  MoveL 9043 to (510.41, 540.16, 160) mm, rotated rx 180 ry 0 rz 160 deg; joints [10.972, 56.166, -5.021, -142.378, 57.459, 157.483]
  Set speed (17.1 mm/s)
  Call Extruder(1063.40800)
  MoveL 9044 to (509.43, 540.4, 160) mm, rotated rx -180 ry 0 rz 160 deg; joints [11.024, 56.007, -4.715, -142.378, 57.595, 157.558]
  Set speed (17.1 mm/s)
  Call Extruder(1069.01822)
  MoveL 9045 to (507.77, 540.76, 160) mm, rotated rx 180 ry 0 rz 160 deg; joints [11.105, 55.733, -4.19, -142.385, 57.825, 157.692]
  Call Extruder(1074.68107)
  MoveL 9046 to (506.08, 541.04, 160) mm, rotated rx 180 ry 0 rz 160 deg; joints [11.18, 55.455, -3.655, -142.401, 58.057, 157.833]
  Call Extruder(1080.09055)
  MoveL 9047 to (504.45, 541.25, 160) mm, rotated rx 180 ry 0 rz 160 deg; joints [11.245, 55.187, -3.141, -142.425, 58.276, 157.973]
  Set speed (17.1 mm/s)
  Call Extruder(1085.82019)
  MoveL 9048 to (502.71, 541.4, 160) mm, rotated rx -180 ry 0 rz 160 deg; joints [11.305, 54.901, -2.592, -142.458, 58.507, 158.127]
  Set speed (17.1 mm/s)
  Call Extruder(1091.48567)
  MoveL 9049 to (501, 541.48, 160) mm, rotated rx -180 ry 0 rz 160 deg; joints [11.357, 54.617, -2.047, -142.499, 58.734, 158.284]
  Set speed (17.1 mm/s)
  Call Extruder(1096.89132)
  MoveL 9050 to (499.36, 541.49, 160) mm, rotated rx -180 ry 0 rz 160 deg; joints [11.398, 54.346, -1.526, -142.546, 58.947, 158.438]
  Set speed (10.0 mm/s)
  MoveL 9051 to (499.36, 541.49, 164) mm, rotated rx 180 ry 0 rz 160 deg; joints [11.398, 53.788, -1.416, -142.38, 58.592, 158.119]
  Set speed (120.0 mm/s)
  MoveL 9052 to (500.97, 540.23, 164) mm, rotated rx -180 ry 0 rz 160 deg; joints [11.204, 54.015, -1.85, -142.513, 58.356, 158.081]
  Set speed (17.3 mm/s)
  Call Extruder(1102.39668)
  MoveL 9053 to (499.29, 540.24, 164) mm, rotated rx 180 ry 0 rz 160 deg; joints [11.246, 53.735, -1.315, -142.564, 58.573, 158.239]
  Call Extruder(1107.72599)
  MoveL 9054 to (497.66, 540.17, 164) mm, rotated rx 180 ry 0 rz 160 deg; joints [11.278, 53.463, -0.796, -142.62, 58.781, 158.397]
  Set speed (17.2 mm/s)
  Call Extruder(1113.18708)
  MoveL 9055 to (496, 540.04, 164) mm, rotated rx -180 ry 0 rz 160 deg; joints [11.303, 53.185, -0.265, -142.685, 58.991, 158.562]
  Call Extruder(1118.52641)
  MoveL 9056 to (494.38, 539.85, 164) mm, rotated rx -180 ry 0 rz 160 deg; joints [11.319, 52.913, 0.253, -142.758, 59.193, 158.727]
  Set speed (17.3 mm/s)
  Call Extruder(1123.71666)
  MoveL 9057 to (492.81, 539.59, 164) mm, rotated rx -180 ry 0 rz 160 deg; joints [11.326, 52.65, 0.755, -142.835, 59.387, 158.891]
  Call Extruder(1129.28278)
  MoveL 9058 to (491.14, 539.26, 164) mm, rotated rx -180 ry 0 rz 160 deg; joints [11.326, 52.369, 1.291, -142.926, 59.59, 159.07]
  Set speed (17.2 mm/s)
  Call Extruder(1134.66464)
  MoveL 9059 to (489.55, 538.86, 164) mm, rotated rx 180 ry 0 rz 160 deg; joints [11.317, 52.1, 1.806, -143.022, 59.782, 159.246]
  Set speed (17.2 mm/s)
  Call Extruder(1139.87147)
  MoveL 9060 to (488.02, 538.42, 164) mm, rotated rx -180 ry 0 rz 160 deg; joints [11.299, 51.841, 2.299, -143.123, 59.964, 159.419]
  Set speed (17.2 mm/s)
  Call Extruder(1145.48231)
  MoveL 9061 to (486.39, 537.87, 164) mm, rotated rx 180 ry 0 rz 160 deg; joints [11.271, 51.565, 2.826, -143.24, 60.155, 159.607]
  Set speed (17.2 mm/s)
  Call Extruder(1150.53984)
  MoveL 9062 to (484.95, 537.32, 164) mm, rotated rx 180 ry 0 rz 160 deg; joints [11.238, 51.319, 3.296, -143.352, 60.322, 159.779]
  Set speed (17.2 mm/s)
  Call Extruder(1155.86729)
  MoveL 9063 to (483.45, 536.68, 164) mm, rotated rx 180 ry 0 rz 160 deg; joints [11.195, 51.063, 3.784, -143.478, 60.494, 159.962]
  Set speed (17.3 mm/s)
  Call Extruder(1159.63536)
  MoveL 9064 to (482.41, 536.2, 164) mm, rotated rx 180 ry 0 rz 160 deg; joints [11.159, 50.884, 4.127, -143.571, 60.613, 160.092]
  Call Extruder(1164.11046)
  MoveL 9065 to (481.19, 535.58, 164) mm, rotated rx 180 ry 0 rz 160 deg; joints [11.11, 50.674, 4.527, -143.688, 60.75, 160.247]
  Set speed (17.3 mm/s)
  Call Extruder(1166.72011)
  MoveL 9066 to (480.49, 535.2, 164) mm, rotated rx 180 ry 0 rz 160 deg; joints [11.079, 50.553, 4.758, -143.757, 60.828, 160.338]
  Call Extruder(1169.33186)
  MoveL 9067 to (479.79, 534.8, 164) mm, rotated rx 180 ry 0 rz 160 deg; joints [11.046, 50.433, 4.987, -143.829, 60.905, 160.429]
  Set speed (17.2 mm/s)
  Call Extruder(1172.31752)
  MoveL 9068 to (479.01, 534.33, 164) mm, rotated rx 180 ry 0 rz 160 deg; joints [11.005, 50.297, 5.246, -143.913, 60.991, 160.534]
  Set speed (17.3 mm/s)
  Call Extruder(1175.98709)
  MoveL 9069 to (478.06, 533.74, 164) mm, rotated rx 180 ry 0 rz 160 deg; joints [10.952, 50.132, 5.561, -144.019, 61.095, 160.662]
  Call Extruder(1180.42460)
  MoveL 9070 to (476.94, 532.98, 164) mm, rotated rx 180 ry 0 rz 160 deg; joints [10.882, 49.936, 5.935, -144.153, 61.216, 160.818]
  Set speed (17.2 mm/s)
  Call Extruder(1183.09673)
  MoveL 9071 to (476.27, 532.5, 164) mm, rotated rx -180 ry 0 rz 160 deg; joints [10.836, 49.82, 6.157, -144.235, 61.287, 160.912]
  Set speed (17.2 mm/s)
  Call Extruder(1185.65152)
  MoveL 9072 to (475.65, 532.04, 164) mm, rotated rx -180 ry 0 rz 160 deg; joints [10.791, 49.71, 6.367, -144.316, 61.353, 161.002]
  Set speed (17.2 mm/s)
  Call Extruder(1188.25211)
  MoveL 9073 to (475.02, 531.55, 164) mm, rotated rx -180 ry 0 rz 160 deg; joints [10.744, 49.6, 6.578, -144.399, 61.419, 161.093]
  Set speed (17.2 mm/s)
  Call Extruder(1191.21831)
  MoveL 9074 to (474.31, 530.98, 164) mm, rotated rx 180 ry 0 rz 160 deg; joints [10.687, 49.475, 6.815, -144.496, 61.493, 161.197]
  Set speed (17.2 mm/s)
  Call Extruder(1193.83711)
  MoveL 9075 to (473.7, 530.46, 164) mm, rotated rx 180 ry 0 rz 160 deg; joints [10.634, 49.367, 7.021, -144.584, 61.556, 161.289]
  Set speed (17.2 mm/s)
  Call Extruder(1196.39663)
  MoveL 9076 to (473.11, 529.95, 164) mm, rotated rx 180 ry 0 rz 160 deg; joints [10.581, 49.263, 7.22, -144.671, 61.616, 161.379]
  Set speed (17.2 mm/s)
  Call Extruder(1199.09717)
  MoveL 9077 to (472.51, 529.39, 164) mm, rotated rx -180 ry 0 rz 160 deg; joints [10.522, 49.155, 7.427, -144.764, 61.678, 161.473]
  Call Extruder(1201.94180)
  MoveL 9078 to (471.88, 528.79, 164) mm, rotated rx -180 ry 0 rz 160 deg; joints [10.459, 49.042, 7.641, -144.865, 61.741, 161.572]
  Set speed (17.2 mm/s)
  Call Extruder(1207.42131)
  MoveL 9079 to (470.71, 527.59, 164) mm, rotated rx 180 ry 0 rz 160 deg; joints [10.329, 48.832, 8.043, -145.063, 61.857, 161.763]
  Set speed (17.2 mm/s)
  Call Extruder(1209.85171)
  MoveL 9080 to (470.2, 527.05, 164) mm, rotated rx 180 ry 0 rz 160 deg; joints [10.27, 48.74, 8.218, -145.153, 61.906, 161.847]
  Set speed (17.2 mm/s)
  Call Extruder(1212.71687)
  MoveL 9081 to (469.62, 526.39, 164) mm, rotated rx 180 ry 0 rz 160 deg; joints [10.197, 48.635, 8.419, -145.26, 61.963, 161.946]
  Call Extruder(1215.30637)
  MoveL 9082 to (469.11, 525.79, 164) mm, rotated rx 180 ry 0 rz 160 deg; joints [10.129, 48.541, 8.597, -145.359, 62.011, 162.035]
  Set speed (17.2 mm/s)
  Call Extruder(1217.99933)
  MoveL 9083 to (468.59, 525.15, 164) mm, rotated rx -180 ry 0 rz 160 deg; joints [10.057, 48.446, 8.78, -145.463, 62.061, 162.127]
  Set speed (17.2 mm/s)
  Call Extruder(1220.64109)
  MoveL 9084 to (468.09, 524.52, 164) mm, rotated rx -180 ry 0 rz 160 deg; joints [9.984, 48.354, 8.955, -145.566, 62.107, 162.217]
  Set speed (17.2 mm/s)
  Call Extruder(1223.38075)
  MoveL 9085 to (467.58, 523.85, 164) mm, rotated rx -180 ry 0 rz 160 deg; joints [9.907, 48.261, 9.132, -145.675, 62.153, 162.31]
  Set speed (17.2 mm/s)
  Call Extruder(1226.20172)
  MoveL 9086 to (467.08, 523.15, 164) mm, rotated rx -180 ry 0 rz 160 deg; joints [9.825, 48.168, 9.311, -145.788, 62.199, 162.406]
  Set speed (17.3 mm/s)
  Call Extruder(1228.73103)
  MoveL 9087 to (466.64, 522.51, 164) mm, rotated rx 180 ry 0 rz 160 deg; joints [9.75, 48.086, 9.467, -145.891, 62.238, 162.491]
  Set speed (17.3 mm/s)
  Call Extruder(1231.44468)
  MoveL 9088 to (466.19, 521.82, 164) mm, rotated rx 180 ry 0 rz 160 deg; joints [9.668, 48, 9.631, -146.003, 62.278, 162.581]
  Set speed (17.2 mm/s)
  Call Extruder(1234.06972)
  MoveL 9089 to (465.76, 521.14, 164) mm, rotated rx 180 ry 0 rz 160 deg; joints [9.587, 47.919, 9.786, -146.112, 62.315, 162.668]
  Call Extruder(1236.82307)
  MoveL 9090 to (465.32, 520.42, 164) mm, rotated rx -180 ry 0 rz 160 deg; joints [9.499, 47.836, 9.944, -146.228, 62.351, 162.759]
  Set speed (17.3 mm/s)
  Call Extruder(1239.50905)
  MoveL 9091 to (464.92, 519.71, 164) mm, rotated rx -180 ry 0 rz 160 deg; joints [9.413, 47.757, 10.094, -146.342, 62.385, 162.847]
  Set speed (17.2 mm/s)
  Call Extruder(1242.30123)
  MoveL 9092 to (464.5, 518.96, 164) mm, rotated rx -180 ry 0 rz 160 deg; joints [9.321, 47.678, 10.246, -146.461, 62.418, 162.938]
  Set speed (17.2 mm/s)
  Call Extruder(1244.88259)
  MoveL 9093 to (464.14, 518.26, 164) mm, rotated rx 180 ry 0 rz 160 deg; joints [9.235, 47.607, 10.381, -146.573, 62.447, 163.021]
  Set speed (17.3 mm/s)
  Call Extruder(1247.52606)
  MoveL 9094 to (463.78, 517.54, 164) mm, rotated rx 180 ry 0 rz 160 deg; joints [9.145, 47.536, 10.516, -146.689, 62.474, 163.106]
  Set speed (17.2 mm/s)
  Call Extruder(1252.88420)
  MoveL 9095 to (463.09, 516.05, 164) mm, rotated rx -180 ry 0 rz 160 deg; joints [8.958, 47.4, 10.777, -146.925, 62.524, 163.276]
  Set speed (17.2 mm/s)
  Call Extruder(1258.25337)
  MoveL 9096 to (462.47, 514.53, 164) mm, rotated rx -180 ry 0 rz 160 deg; joints [8.765, 47.273, 11.019, -147.166, 62.566, 163.442]
  Set speed (17.2 mm/s)
  Call Extruder(1263.67576)
  MoveL 9097 to (461.91, 512.98, 164) mm, rotated rx 180 ry 0 rz 160 deg; joints [8.565, 47.154, 11.245, -147.413, 62.599, 163.608]
  Call Extruder(1269.06660)
  MoveL 9098 to (461.41, 511.41, 164) mm, rotated rx 180 ry 0 rz 160 deg; joints [8.361, 47.046, 11.452, -147.66, 62.625, 163.768]
  Set speed (17.2 mm/s)
  Call Extruder(1274.56925)
  MoveL 9099 to (460.97, 509.78, 164) mm, rotated rx 180 ry 0 rz 160 deg; joints [8.148, 46.946, 11.642, -147.916, 62.643, 163.929]
  Set speed (17.2 mm/s)
  Call Extruder(1279.89206)
  MoveL 9100 to (460.6, 508.2, 164) mm, rotated rx -180 ry 0 rz 160 deg; joints [7.938, 46.86, 11.807, -148.165, 62.651, 164.08]
  Set speed (17.3 mm/s)
  Call Extruder(1285.41223)
  MoveL 9101 to (460.29, 506.54, 164) mm, rotated rx -180 ry 0 rz 160 deg; joints [7.717, 46.781, 11.958, -148.424, 62.652, 164.233]
  Call Extruder(1290.88446)
  MoveL 9102 to (460.06, 504.88, 164) mm, rotated rx -180 ry 0 rz 160 deg; joints [7.493, 46.714, 12.086, -148.683, 62.644, 164.38]
  Set speed (17.2 mm/s)
  Call Extruder(1296.18613)
  MoveL 9103 to (459.89, 503.27, 164) mm, rotated rx -180 ry 0 rz 160 deg; joints [7.274, 46.659, 12.191, -148.934, 62.627, 164.518]
  Set speed (17.3 mm/s)
  Call Extruder(1301.69852)
  MoveL 9104 to (459.79, 501.59, 164) mm, rotated rx 180 ry 0 rz 160 deg; joints [7.044, 46.613, 12.279, -149.195, 62.602, 164.657]
  Set speed (17.2 mm/s)
  Call Extruder(1306.85050)
  MoveL 9105 to (459.75, 500.02, 164) mm, rotated rx -180 ry 0 rz 160 deg; joints [6.827, 46.579, 12.342, -149.438, 62.571, 164.783]
  Call Extruder(1311.56706)
  MoveL 9106 to (459.78, 498.58, 164) mm, rotated rx 180 ry 0 rz 160 deg; joints [6.628, 46.559, 12.381, -149.66, 62.535, 164.894]
  Call Extruder(1316.68940)
  MoveL 9107 to (459.87, 497.01, 164) mm, rotated rx 180 ry 0 rz 160 deg; joints [6.41, 46.545, 12.408, -149.9, 62.489, 165.01]
  Set speed (17.3 mm/s)
  Call Extruder(1321.58133)
  MoveL 9108 to (460.01, 495.52, 164) mm, rotated rx -180 ry 0 rz 160 deg; joints [6.202, 46.541, 12.415, -150.128, 62.439, 165.117]
  Set speed (17.3 mm/s)
  Call Extruder(1326.10523)
  MoveL 9109 to (460.19, 494.15, 164) mm, rotated rx 180 ry 0 rz 160 deg; joints [6.01, 46.546, 12.406, -150.337, 62.386, 165.212]
  Set speed (17.3 mm/s)
  Call Extruder(1331.17816)
  MoveL 9110 to (460.44, 492.62, 164) mm, rotated rx -180 ry 0 rz 160 deg; joints [5.794, 46.56, 12.379, -150.569, 62.32, 165.314]
  Set speed (17.3 mm/s)
  Call Extruder(1335.86329)
  MoveL 9111 to (460.73, 491.22, 164) mm, rotated rx -180 ry 0 rz 160 deg; joints [5.596, 46.582, 12.337, -150.78, 62.252, 165.403]
  Set speed (17.2 mm/s)
  Call Extruder(1340.95386)
  MoveL 9112 to (461.1, 489.71, 164) mm, rotated rx 180 ry 0 rz 160 deg; joints [5.382, 46.615, 12.275, -151.007, 62.173, 165.496]
  Set speed (17.2 mm/s)
  Call Extruder(1345.56843)
  MoveL 9113 to (461.48, 488.35, 164) mm, rotated rx 180 ry 0 rz 160 deg; joints [5.19, 46.653, 12.202, -151.209, 62.094, 165.576]
  Set speed (17.2 mm/s)
  Call Extruder(1350.72526)
  MoveL 9114 to (461.97, 486.85, 164) mm, rotated rx 180 ry 0 rz 160 deg; joints [4.976, 46.705, 12.103, -151.431, 62, 165.66]
  Set speed (17.2 mm/s)
  Call Extruder(1355.73817)
  MoveL 9115 to (462.5, 485.41, 164) mm, rotated rx 180 ry 0 rz 160 deg; joints [4.771, 46.765, 11.989, -151.642, 61.901, 165.737]
  Call Extruder(1360.34080)
  MoveL 9116 to (463.03, 484.11, 164) mm, rotated rx 180 ry 0 rz 160 deg; joints [4.585, 46.828, 11.869, -151.832, 61.805, 165.802]
  Set speed (17.3 mm/s)
  Call Extruder(1365.27188)
  MoveL 9117 to (463.65, 482.74, 164) mm, rotated rx 180 ry 0 rz 160 deg; joints [4.389, 46.904, 11.723, -152.03, 61.696, 165.867]
  Set speed (17.2 mm/s)
  Call Extruder(1369.73169)
  MoveL 9118 to (464.26, 481.52, 164) mm, rotated rx 180 ry 0 rz 160 deg; joints [4.214, 46.98, 11.578, -152.205, 61.592, 165.922]
  Set speed (17.2 mm/s)
  Call Extruder(1374.93959)
  MoveL 9119 to (465.01, 480.12, 164) mm, rotated rx 180 ry 0 rz 160 deg; joints [4.014, 47.078, 11.391, -152.404, 61.465, 165.98]
  Set speed (17.2 mm/s)
  Call Extruder(1379.75206)
  MoveL 9120 to (465.76, 478.85, 164) mm, rotated rx 180 ry 0 rz 160 deg; joints [3.833, 47.176, 11.203, -152.581, 61.342, 166.029]
  Call Extruder(1384.92062)
  MoveL 9121 to (466.62, 477.52, 164) mm, rotated rx 180 ry 0 rz 160 deg; joints [3.643, 47.291, 10.984, -152.766, 61.204, 166.076]
  Call Extruder(1389.45717)
  MoveL 9122 to (467.41, 476.39, 164) mm, rotated rx -180 ry 0 rz 160 deg; joints [3.481, 47.399, 10.778, -152.921, 61.077, 166.111]
  Set speed (17.2 mm/s)
  Call Extruder(1394.19668)
  MoveL 9123 to (468.28, 475.23, 164) mm, rotated rx 180 ry 0 rz 160 deg; joints [3.315, 47.519, 10.549, -153.077, 60.94, 166.144]
  Call Extruder(1399.13732)
  MoveL 9124 to (469.23, 474.06, 164) mm, rotated rx 180 ry 0 rz 160 deg; joints [3.148, 47.652, 10.295, -153.233, 60.792, 166.172]
  Set speed (17.3 mm/s)
  Call Extruder(1403.98459)
  MoveL 9125 to (470.21, 472.94, 164) mm, rotated rx -180 ry 0 rz 160 deg; joints [2.988, 47.79, 10.032, -153.379, 60.642, 166.194]
  Set speed (17.3 mm/s)
  Call Extruder(1408.72195)
  MoveL 9126 to (471.2, 471.89, 164) mm, rotated rx 180 ry 0 rz 160 deg; joints [2.838, 47.932, 9.762, -153.514, 60.491, 166.21]
  Set speed (17.3 mm/s)
  Call Extruder(1413.62945)
  MoveL 9127 to (472.27, 470.84, 164) mm, rotated rx 180 ry 0 rz 160 deg; joints [2.688, 48.086, 9.468, -153.646, 60.33, 166.222]
  Set speed (17.2 mm/s)
  Call Extruder(1418.25129)
  MoveL 9128 to (473.31, 469.88, 164) mm, rotated rx 180 ry 0 rz 160 deg; joints [2.552, 48.237, 9.179, -153.763, 60.175, 166.227]
  Call Extruder(1423.26639)
  MoveL 9129 to (474.48, 468.88, 164) mm, rotated rx 180 ry 0 rz 160 deg; joints [2.411, 48.408, 8.853, -153.882, 60.002, 166.227]
  Call Extruder(1428.06443)
  MoveL 9130 to (475.63, 467.97, 164) mm, rotated rx 180 ry 0 rz 160 deg; joints [2.282, 48.577, 8.529, -153.988, 59.832, 166.221]
  Call Extruder(1433.02690)
  MoveL 9131 to (476.86, 467.08, 164) mm, rotated rx 180 ry 0 rz 160 deg; joints [2.155, 48.76, 8.181, -154.088, 59.653, 166.209]
  Set speed (17.3 mm/s)
  Call Extruder(1437.79644)
  MoveL 9132 to (478.06, 466.26, 164) mm, rotated rx 180 ry 0 rz 160 deg; joints [2.04, 48.941, 7.835, -154.176, 59.478, 166.191]
  Set speed (17.3 mm/s)
  Call Extruder(1442.40095)
  MoveL 9133 to (479.26, 465.52, 164) mm, rotated rx -180 ry 0 rz 160 deg; joints [1.934, 49.121, 7.492, -154.252, 59.305, 166.169]
  Set speed (17.3 mm/s)
  Call Extruder(1447.50015)
  MoveL 9134 to (480.61, 464.74, 164) mm, rotated rx -180 ry 0 rz 160 deg; joints [1.825, 49.326, 7.1, -154.329, 59.111, 166.139]
  Set speed (17.2 mm/s)
  Call Extruder(1453.20412)
  MoveL 9135 to (482.15, 463.93, 164) mm, rotated rx 180 ry 0 rz 160 deg; joints [1.711, 49.562, 6.65, -154.401, 58.891, 166.097]
  Set speed (17.2 mm/s)
  Call Extruder(1457.17333)
  MoveL 9136 to (483.25, 463.41, 164) mm, rotated rx 180 ry 0 rz 160 deg; joints [1.638, 49.73, 6.329, -154.444, 58.735, 166.062]
  Set speed (17.2 mm/s)
  Call Extruder(1461.95242)
  MoveL 9137 to (484.59, 462.83, 164) mm, rotated rx -180 ry 0 rz 160 deg; joints [1.556, 49.937, 5.934, -154.488, 58.545, 166.016]
  Set speed (17.3 mm/s)
  Call Extruder(1466.98216)
  MoveL 9138 to (486.02, 462.27, 164) mm, rotated rx -180 ry 0 rz 160 deg; joints [1.477, 50.16, 5.509, -154.525, 58.344, 165.961]
  Set speed (17.2 mm/s)
  Call Extruder(1471.84329)
  MoveL 9139 to (487.42, 461.77, 164) mm, rotated rx -180 ry 0 rz 160 deg; joints [1.408, 50.379, 5.09, -154.55, 58.147, 165.902]
  Call Extruder(1476.74031)
  MoveL 9140 to (488.85, 461.33, 164) mm, rotated rx 180 ry 0 rz 160 deg; joints [1.346, 50.604, 4.661, -154.567, 57.947, 165.836]
  Set speed (17.3 mm/s)
  Call Extruder(1481.51368)
  MoveL 9141 to (490.26, 460.96, 164) mm, rotated rx -180 ry 0 rz 160 deg; joints [1.292, 50.827, 4.235, -154.573, 57.751, 165.766]
  Set speed (17.3 mm/s)
  Call Extruder(1486.28147)
  MoveL 9142 to (491.68, 460.63, 164) mm, rotated rx 180 ry 0 rz 160 deg; joints [1.245, 51.053, 3.804, -154.571, 57.554, 165.69]
  Set speed (17.3 mm/s)
  Call Extruder(1490.95394)
  MoveL 9143 to (493.08, 460.36, 164) mm, rotated rx 180 ry 0 rz 160 deg; joints [1.206, 51.277, 3.375, -154.56, 57.36, 165.61]
  Set speed (17.3 mm/s)
  Call Extruder(1496.06278)
  MoveL 9144 to (494.63, 460.12, 164) mm, rotated rx 180 ry 0 rz 160 deg; joints [1.171, 51.526, 2.902, -154.538, 57.148, 165.517]
  Set speed (17.2 mm/s)
  Call Extruder(1500.87565)
  MoveL 9145 to (496.09, 459.95, 164) mm, rotated rx 180 ry 0 rz 160 deg; joints [1.146, 51.762, 2.451, -154.507, 56.948, 165.423]
  Set speed (17.2 mm/s)
  Call Extruder(1505.77291)
  MoveL 9146 to (497.58, 459.83, 164) mm, rotated rx -180 ry 0 rz 160 deg; joints [1.127, 52.005, 1.987, -154.468, 56.744, 165.321]
  Set speed (17.3 mm/s)
  Call Extruder(1510.56917)
  MoveL 9147 to (499.05, 459.77, 164) mm, rotated rx -180 ry 0 rz 160 deg; joints [1.115, 52.244, 1.53, -154.419, 56.544, 165.216]
  Set speed (17.3 mm/s)
  Call Extruder(1515.26906)
  MoveL 9148 to (500.48, 459.76, 164) mm, rotated rx 180 ry 0 rz 160 deg; joints [1.11, 52.48, 1.079, -154.363, 56.35, 165.108]
  Call Extruder(1520.34091)
  MoveL 9149 to (502.03, 459.81, 164) mm, rotated rx -180 ry 0 rz 160 deg; joints [1.113, 52.737, 0.59, -154.293, 56.14, 164.985]
  Set speed (17.3 mm/s)
  Call Extruder(1525.13170)
  MoveL 9150 to (503.49, 459.91, 164) mm, rotated rx 180 ry 0 rz 160 deg; joints [1.122, 52.98, 0.125, -154.217, 55.944, 164.863]
  Set speed (17.2 mm/s)
  Call Extruder(1529.97241)
  MoveL 9151 to (504.96, 460.07, 164) mm, rotated rx -180 ry 0 rz 160 deg; joints [1.138, 53.226, -0.344, -154.133, 55.746, 164.735]
  Set speed (17.2 mm/s)
  Call Extruder(1534.57519)
  MoveL 9152 to (506.36, 460.26, 164) mm, rotated rx -180 ry 0 rz 160 deg; joints [1.159, 53.461, -0.792, -154.044, 55.561, 164.608]
  Set speed (17.2 mm/s)
  Call Extruder(1539.34961)
  MoveL 9153 to (507.79, 460.52, 164) mm, rotated rx 180 ry 0 rz 160 deg; joints [1.188, 53.704, -1.256, -153.944, 55.37, 164.472]
  Set speed (17.3 mm/s)
  Call Extruder(1544.52807)
  MoveL 9154 to (509.34, 460.86, 164) mm, rotated rx -180 ry 0 rz 160 deg; joints [1.226, 53.968, -1.759, -153.827, 55.165, 164.318]
  Set speed (17.3 mm/s)
  Call Extruder(1549.38509)
  MoveL 9155 to (510.78, 461.23, 164) mm, rotated rx 180 ry 0 rz 160 deg; joints [1.268, 54.214, -2.23, -153.708, 54.975, 164.169]
  Set speed (17.3 mm/s)
  Call Extruder(1554.03460)
  MoveL 9156 to (512.14, 461.63, 164) mm, rotated rx 180 ry 0 rz 160 deg; joints [1.315, 54.45, -2.679, -153.586, 54.796, 164.021]
  Set speed (17.3 mm/s)
  Call Extruder(1558.96594)
  MoveL 9157 to (513.57, 462.12, 164) mm, rotated rx 180 ry 0 rz 160 deg; joints [1.37, 54.698, -3.153, -153.449, 54.61, 163.86]
  Call Extruder(1563.55660)
  MoveL 9158 to (514.88, 462.61, 164) mm, rotated rx -180 ry 0 rz 160 deg; joints [1.428, 54.928, -3.591, -153.315, 54.439, 163.706]
  Set speed (17.3 mm/s)
  Call Extruder(1568.65646)
  MoveL 9159 to (516.32, 463.22, 164) mm, rotated rx -180 ry 0 rz 160 deg; joints [1.498, 55.181, -4.075, -153.158, 54.254, 163.531]
  Call Extruder(0.00000)
  Set speed (17.3 mm/s)
  Call Extruder(4.61765)
  MoveL 9160 to (517.6, 463.81, 164) mm, rotated rx 180 ry 0 rz 160 deg; joints [1.567, 55.408, -4.509, -153.01, 54.089, 163.368]
  Set speed (17.3 mm/s)
  Call Extruder(9.77849)
  MoveL 9161 to (519.01, 464.53, 164) mm, rotated rx -180 ry 0 rz 160 deg; joints [1.65, 55.66, -4.988, -152.836, 53.91, 163.182]
  Set speed (17.3 mm/s)
  Call Extruder(14.71469)
  MoveL 9162 to (520.32, 465.27, 164) mm, rotated rx -180 ry 0 rz 160 deg; joints [1.735, 55.897, -5.44, -152.662, 53.744, 163]
  Call Extruder(19.28491)
  MoveL 9163 to (521.52, 466, 164) mm, rotated rx 180 ry 0 rz 160 deg; joints [1.819, 56.113, -5.853, -152.496, 53.594, 162.828]
  Set speed (17.3 mm/s)
  Call Extruder(24.21319)
  MoveL 9164 to (522.77, 466.82, 164) mm, rotated rx -180 ry 0 rz 160 deg; joints [1.915, 56.343, -6.292, -152.311, 53.437, 162.64]
  Set speed (17.3 mm/s)
  Call Extruder(28.89791)
  MoveL 9165 to (523.94, 467.66, 164) mm, rotated rx 180 ry 0 rz 160 deg; joints [2.011, 56.558, -6.702, -152.129, 53.293, 162.459]
  Set speed (17.3 mm/s)
  Call Extruder(33.82593)
  MoveL 9166 to (525.14, 468.57, 164) mm, rotated rx -180 ry 0 rz 160 deg; joints [2.116, 56.781, -7.126, -151.933, 53.147, 162.266]
  Set speed (17.2 mm/s)
  Call Extruder(38.75984)
  MoveL 9167 to (526.29, 469.54, 164) mm, rotated rx 180 ry 0 rz 160 deg; joints [2.227, 56.998, -7.541, -151.731, 53.007, 162.07]
  Set speed (17.3 mm/s)
  Call Extruder(43.43285)
  MoveL 9168 to (527.36, 470.49, 164) mm, rotated rx 180 ry 0 rz 160 deg; joints [2.336, 57.2, -7.926, -151.535, 52.88, 161.882]
  Set speed (17.3 mm/s)
  Call Extruder(48.58755)
  MoveL 9169 to (528.5, 471.58, 164) mm, rotated rx -180 ry 0 rz 160 deg; joints [2.462, 57.416, -8.339, -151.314, 52.746, 161.674]
  Call Extruder(53.66629)
  MoveL 9170 to (529.57, 472.71, 164) mm, rotated rx 180 ry 0 rz 160 deg; joints [2.59, 57.624, -8.735, -151.092, 52.622, 161.467]
  Set speed (17.3 mm/s)
  Call Extruder(56.40603)
  MoveL 9171 to (530.13, 473.33, 164) mm, rotated rx 180 ry 0 rz 160 deg; joints [2.661, 57.733, -8.944, -150.97, 52.558, 161.355]
  Set speed (17.2 mm/s)
  Call Extruder(59.26622)
  MoveL 9172 to (530.71, 473.99, 164) mm, rotated rx 180 ry 0 rz 160 deg; joints [2.737, 57.846, -9.158, -150.842, 52.493, 161.238]
  Set speed (17.2 mm/s)
  Call Extruder(61.81879)
  MoveL 9173 to (531.2, 474.59, 164) mm, rotated rx 180 ry 0 rz 160 deg; joints [2.805, 57.944, -9.345, -150.727, 52.437, 161.133]
  Set speed (17.2 mm/s)
  Call Extruder(64.41399)
  MoveL 9174 to (531.7, 475.21, 164) mm, rotated rx 180 ry 0 rz 160 deg; joints [2.876, 58.042, -9.532, -150.609, 52.383, 161.026]
  Call Extruder(67.13695)
  MoveL 9175 to (532.21, 475.87, 164) mm, rotated rx -180 ry 0 rz 160 deg; joints [2.951, 58.143, -9.725, -150.484, 52.327, 160.915]
  Set speed (17.2 mm/s)
  Call Extruder(69.90550)
  MoveL 9176 to (532.7, 476.55, 164) mm, rotated rx 180 ry 0 rz 160 deg; joints [3.029, 58.243, -9.917, -150.356, 52.274, 160.801]
  Call Extruder(72.52977)
  MoveL 9177 to (533.16, 477.21, 164) mm, rotated rx 180 ry 0 rz 160 deg; joints [3.104, 58.337, -10.095, -150.235, 52.225, 160.693]
  Call Extruder(78.09547)
  MoveL 9178 to (534.1, 478.63, 164) mm, rotated rx -180 ry 0 rz 160 deg; joints [3.266, 58.528, -10.459, -149.974, 52.128, 160.465]
  Set speed (17.2 mm/s)
  Call Extruder(82.89360)
  MoveL 9179 to (534.86, 479.88, 164) mm, rotated rx 180 ry 0 rz 160 deg; joints [3.409, 58.685, -10.759, -149.748, 52.053, 160.27]
  Set speed (17.2 mm/s)
  Call Extruder(87.82933)
  MoveL 9180 to (535.58, 481.2, 164) mm, rotated rx -180 ry 0 rz 160 deg; joints [3.559, 58.839, -11.052, -149.514, 51.983, 160.07]
  Set speed (17.2 mm/s)
  Call Extruder(91.41981)
  MoveL 9181 to (536.08, 482.18, 164) mm, rotated rx -180 ry 0 rz 160 deg; joints [3.67, 58.946, -11.256, -149.342, 51.938, 159.926]
  Set speed (17.2 mm/s)
  Call Extruder(94.08306)
  MoveL 9182 to (536.43, 482.91, 164) mm, rotated rx 180 ry 0 rz 160 deg; joints [3.754, 59.023, -11.402, -149.215, 51.907, 159.819]
  Set speed (17.2 mm/s)
  Call Extruder(96.97442)
  MoveL 9183 to (536.8, 483.71, 164) mm, rotated rx 180 ry 0 rz 160 deg; joints [3.845, 59.103, -11.556, -149.076, 51.876, 159.704]
  Set speed (17.2 mm/s)
  Call Extruder(102.36922)
  MoveL 9184 to (537.43, 485.23, 164) mm, rotated rx 180 ry 0 rz 160 deg; joints [4.018, 59.245, -11.827, -148.818, 51.826, 159.492]
  Set speed (17.2 mm/s)
  Call Extruder(107.64359)
  MoveL 9185 to (538, 486.74, 164) mm, rotated rx 180 ry 0 rz 160 deg; joints [4.19, 59.374, -12.073, -148.565, 51.786, 159.288]
  Set speed (17.2 mm/s)
  Call Extruder(113.16762)
  MoveL 9186 to (538.52, 488.35, 164) mm, rotated rx -180 ry 0 rz 160 deg; joints [4.373, 59.499, -12.31, -148.301, 51.755, 159.078]
  Set speed (17.3 mm/s)
  Call Extruder(118.32270)
  MoveL 9187 to (538.95, 489.87, 164) mm, rotated rx 180 ry 0 rz 160 deg; joints [4.547, 59.605, -12.512, -148.055, 51.736, 158.886]
  Call Extruder(123.83762)
  MoveL 9188 to (539.34, 491.51, 164) mm, rotated rx -180 ry 0 rz 160 deg; joints [4.734, 59.706, -12.706, -147.794, 51.726, 158.686]
  Set speed (17.3 mm/s)
  Call Extruder(129.16621)
  MoveL 9189 to (539.65, 493.11, 164) mm, rotated rx 180 ry 0 rz 160 deg; joints [4.917, 59.793, -12.871, -147.544, 51.726, 158.498]
  Set speed (17.2 mm/s)
  Call Extruder(134.76605)
  MoveL 9190 to (539.9, 494.8, 164) mm, rotated rx 180 ry 0 rz 160 deg; joints [5.111, 59.872, -13.023, -147.283, 51.737, 158.306]
  Set speed (17.2 mm/s)
  Call Extruder(140.24021)
  MoveL 9191 to (540.09, 496.46, 164) mm, rotated rx 180 ry 0 rz 160 deg; joints [5.302, 59.938, -13.147, -147.032, 51.758, 158.125]
  Set speed (17.3 mm/s)
  Call Extruder(145.52557)
  MoveL 9192 to (540.2, 498.07, 164) mm, rotated rx 180 ry 0 rz 160 deg; joints [5.488, 59.989, -13.245, -146.792, 51.789, 157.957]
  Set speed (17.3 mm/s)
  Call Extruder(150.71373)
  MoveL 9193 to (540.24, 499.66, 164) mm, rotated rx 180 ry 0 rz 160 deg; joints [5.672, 60.028, -13.32, -146.561, 51.828, 157.799]
  Set speed (17.3 mm/s)
  Call Extruder(156.30675)
  MoveL 9194 to (540.22, 501.37, 164) mm, rotated rx -180 ry 0 rz 160 deg; joints [5.87, 60.058, -13.376, -146.316, 51.881, 157.636]
  Set speed (17.2 mm/s)
  Call Extruder(161.64443)
  MoveL 9195 to (540.13, 503, 164) mm, rotated rx 180 ry 0 rz 160 deg; joints [6.06, 60.074, -13.407, -146.087, 51.941, 157.488]
  Call Extruder(167.06757)
  MoveL 9196 to (539.97, 504.65, 164) mm, rotated rx 180 ry 0 rz 160 deg; joints [6.253, 60.078, -13.414, -145.859, 52.012, 157.346]
  Set speed (17.3 mm/s)
  Call Extruder(172.42728)
  MoveL 9197 to (539.75, 506.27, 164) mm, rotated rx 180 ry 0 rz 160 deg; joints [6.443, 60.07, -13.399, -145.639, 52.092, 157.214]
  Call Extruder(177.54201)
  MoveL 9198 to (539.48, 507.81, 164) mm, rotated rx 180 ry 0 rz 160 deg; joints [6.625, 60.051, -13.362, -145.434, 52.177, 157.096]
  Set speed (17.3 mm/s)
  Call Extruder(183.16286)
  MoveL 9199 to (539.11, 509.49, 164) mm, rotated rx 180 ry 0 rz 160 deg; joints [6.824, 60.017, -13.298, -145.216, 52.28, 156.976]
  Set speed (17.3 mm/s)
  Call Extruder(189.03860)
  MoveL 9200 to (538.65, 511.23, 164) mm, rotated rx -180 ry 0 rz 160 deg; joints [7.032, 59.969, -13.207, -144.994, 52.396, 156.86]
  Set speed (17.3 mm/s)
  Call Extruder(193.69971)
  MoveL 9201 to (538.22, 512.59, 164) mm, rotated rx 180 ry 0 rz 160 deg; joints [7.195, 59.919, -13.111, -144.825, 52.498, 156.778]
  Set speed (17.3 mm/s)
  Call Extruder(199.08064)
  MoveL 9202 to (537.68, 514.14, 164) mm, rotated rx -180 ry 0 rz 160 deg; joints [7.383, 59.851, -12.982, -144.635, 52.623, 156.691]
  Set speed (17.2 mm/s)
  Call Extruder(204.66454)
  MoveL 9203 to (537.04, 515.72, 164) mm, rotated rx -180 ry 0 rz 160 deg; joints [7.576, 59.768, -12.825, -144.445, 52.76, 156.61]
  Set speed (17.3 mm/s)
  Call Extruder(209.82660)
  MoveL 9204 to (536.4, 517.16, 164) mm, rotated rx -180 ry 0 rz 160 deg; joints [7.753, 59.681, -12.658, -144.276, 52.894, 156.545]
  Set speed (17.3 mm/s)
  Call Extruder(212.76425)
  MoveL 9205 to (536.01, 517.97, 164) mm, rotated rx -180 ry 0 rz 160 deg; joints [7.853, 59.626, -12.554, -144.184, 52.974, 156.512]
  Set speed (17.2 mm/s)
  Call Extruder(215.42753)
  MoveL 9206 to (535.63, 518.7, 164) mm, rotated rx -180 ry 0 rz 160 deg; joints [7.942, 59.574, -12.453, -144.102, 53.049, 156.485]
  Set speed (17.2 mm/s)
  Call Extruder(218.19363)
  MoveL 9207 to (535.23, 519.44, 164) mm, rotated rx 180 ry 0 rz 160 deg; joints [8.035, 59.517, -12.345, -144.018, 53.128, 156.459]
  Call Extruder(220.87107)
  MoveL 9208 to (534.83, 520.15, 164) mm, rotated rx -180 ry 0 rz 160 deg; joints [8.124, 59.459, -12.235, -143.939, 53.206, 156.436]
  Call Extruder(223.51382)
  MoveL 9209 to (534.42, 520.85, 164) mm, rotated rx -180 ry 0 rz 160 deg; joints [8.212, 59.4, -12.121, -143.862, 53.284, 156.416]
  Set speed (17.2 mm/s)
  Call Extruder(226.01827)
  MoveL 9210 to (534.02, 521.5, 164) mm, rotated rx 180 ry 0 rz 160 deg; joints [8.294, 59.34, -12.008, -143.792, 53.361, 156.399]
  Call Extruder(230.46743)
  MoveL 9211 to (533.27, 522.63, 164) mm, rotated rx 180 ry 0 rz 160 deg; joints [8.439, 59.229, -11.797, -143.671, 53.5, 156.375]
  Set speed (17.3 mm/s)
  Call Extruder(234.10450)
  MoveL 9212 to (532.63, 523.55, 164) mm, rotated rx 180 ry 0 rz 160 deg; joints [8.556, 59.134, -11.615, -143.576, 53.616, 156.36]
  Set speed (17.3 mm/s)
  Call Extruder(236.82504)
  MoveL 9213 to (532.14, 524.22, 164) mm, rotated rx 180 ry 0 rz 160 deg; joints [8.642, 59.06, -11.473, -143.507, 53.705, 156.351]
  Set speed (17.2 mm/s)
  Call Extruder(239.67627)
  MoveL 9214 to (531.61, 524.91, 164) mm, rotated rx -180 ry 0 rz 160 deg; joints [8.732, 58.979, -11.319, -143.437, 53.8, 156.345]
  Call Extruder(242.36553)
  MoveL 9215 to (531.09, 525.55, 164) mm, rotated rx -180 ry 0 rz 160 deg; joints [8.816, 58.9, -11.168, -143.373, 53.891, 156.342]
  Set speed (17.2 mm/s)
  Call Extruder(246.49092)
  MoveL 9216 to (530.28, 526.51, 164) mm, rotated rx -180 ry 0 rz 160 deg; joints [8.943, 58.774, -10.929, -143.278, 54.034, 156.341]
  Set speed (17.2 mm/s)
  Call Extruder(251.80850)
  MoveL 9217 to (529.19, 527.71, 164) mm, rotated rx 180 ry 0 rz 160 deg; joints [9.103, 58.605, -10.606, -143.164, 54.221, 156.349]
  Set speed (17.2 mm/s)
  Call Extruder(255.86966)
  MoveL 9218 to (528.32, 528.59, 164) mm, rotated rx -180 ry 0 rz 160 deg; joints [9.223, 58.469, -10.347, -143.082, 54.368, 156.361]
  Set speed (17.3 mm/s)
  Call Extruder(258.43514)
  MoveL 9219 to (527.76, 529.14, 164) mm, rotated rx -180 ry 0 rz 160 deg; joints [9.297, 58.381, -10.178, -143.032, 54.462, 156.371]
  Set speed (17.3 mm/s)
  Call Extruder(261.06836)
  MoveL 9220 to (527.17, 529.69, 164) mm, rotated rx -180 ry 0 rz 160 deg; joints [9.373, 58.288, -10.002, -142.983, 54.559, 156.384]
  Call Extruder(263.80830)
  MoveL 9221 to (526.54, 530.25, 164) mm, rotated rx -180 ry 0 rz 160 deg; joints [9.451, 58.189, -9.814, -142.934, 54.661, 156.399]
  Set speed (17.2 mm/s)
  Call Extruder(266.42764)
  MoveL 9222 to (525.94, 530.77, 164) mm, rotated rx -180 ry 0 rz 160 deg; joints [9.524, 58.093, -9.63, -142.89, 54.76, 156.417]
  Call Extruder(269.15438)
  MoveL 9223 to (525.29, 531.3, 164) mm, rotated rx -180 ry 0 rz 160 deg; joints [9.599, 57.991, -9.435, -142.845, 54.864, 156.437]
  Set speed (17.2 mm/s)
  Call Extruder(272.04094)
  MoveL 9224 to (524.6, 531.85, 164) mm, rotated rx 180 ry 0 rz 160 deg; joints [9.677, 57.881, -9.225, -142.8, 54.975, 156.46]
  Set speed (17.2 mm/s)
  Call Extruder(274.48416)
  MoveL 9225 to (524.01, 532.3, 164) mm, rotated rx -180 ry 0 rz 160 deg; joints [9.742, 57.786, -9.043, -142.764, 55.07, 156.482]
  Set speed (17.3 mm/s)
  Call Extruder(277.27156)
  MoveL 9226 to (523.32, 532.8, 164) mm, rotated rx -180 ry 0 rz 160 deg; joints [9.815, 57.675, -8.833, -142.725, 55.179, 156.51]
  Set speed (17.2 mm/s)
  Call Extruder(280.10604)
  MoveL 9227 to (522.61, 533.29, 164) mm, rotated rx -180 ry 0 rz 160 deg; joints [9.887, 57.561, -8.615, -142.687, 55.29, 156.54]
  Set speed (17.2 mm/s)
  Call Extruder(282.60739)
  MoveL 9228 to (521.97, 533.72, 164) mm, rotated rx -180 ry 0 rz 160 deg; joints [9.95, 57.459, -8.42, -142.656, 55.389, 156.568]
  Set speed (17.2 mm/s)
  Call Extruder(288.02384)
  MoveL 9229 to (520.57, 534.59, 164) mm, rotated rx -180 ry 0 rz 160 deg; joints [10.083, 57.232, -7.988, -142.593, 55.605, 156.636]
  Call Extruder(293.25804)
  MoveL 9230 to (519.17, 535.38, 164) mm, rotated rx 180 ry 0 rz 160 deg; joints [10.206, 57.007, -7.559, -142.542, 55.816, 156.709]
  Call Extruder(296.11447)
  MoveL 9231 to (518.4, 535.79, 164) mm, rotated rx 180 ry 0 rz 160 deg; joints [10.271, 56.882, -7.32, -142.517, 55.931, 156.752]
  Set speed (17.2 mm/s)
  Call Extruder(298.78339)
  MoveL 9232 to (517.67, 536.15, 164) mm, rotated rx -180 ry 0 rz 160 deg; joints [10.33, 56.764, -7.094, -142.495, 56.04, 156.795]
  Set speed (17.2 mm/s)
  Call Extruder(301.48397)
  MoveL 9233 to (516.93, 536.51, 164) mm, rotated rx -180 ry 0 rz 160 deg; joints [10.388, 56.642, -6.863, -142.476, 56.15, 156.839]
  Set speed (17.2 mm/s)
  Call Extruder(307.01749)
  MoveL 9234 to (515.38, 537.19, 164) mm, rotated rx -180 ry 0 rz 160 deg; joints [10.503, 56.39, -6.381, -142.442, 56.377, 156.937]
  Set speed (17.3 mm/s)
  Call Extruder(312.29942)
  MoveL 9235 to (513.88, 537.77, 164) mm, rotated rx 180 ry 0 rz 160 deg; joints [10.606, 56.144, -5.912, -142.418, 56.594, 157.037]
  Set speed (17.2 mm/s)
  Call Extruder(314.67045)
  MoveL 9236 to (513.19, 538.02, 164) mm, rotated rx -180 ry 0 rz 160 deg; joints [10.651, 56.032, -5.699, -142.41, 56.692, 157.084]
  Set speed (17.2 mm/s)
  Call Extruder(317.83568)
  MoveL 9237 to (512.28, 538.33, 164) mm, rotated rx 180 ry 0 rz 160 deg; joints [10.708, 55.882, -5.413, -142.401, 56.822, 157.149]
  Set speed (17.2 mm/s)
  Call Extruder(323.22883)
  MoveL 9238 to (510.7, 538.8, 164) mm, rotated rx -180 ry 0 rz 160 deg; joints [10.801, 55.623, -4.918, -142.393, 57.045, 157.264]
  Set speed (17.3 mm/s)
  Call Extruder(328.63225)
  MoveL 9239 to (509.1, 539.2, 164) mm, rotated rx 180 ry 0 rz 160 deg; joints [10.886, 55.359, -4.415, -142.393, 57.267, 157.387]
  Call Extruder(333.84331)
  MoveL 9240 to (507.54, 539.53, 164) mm, rotated rx 180 ry 0 rz 160 deg; joints [10.962, 55.102, -3.925, -142.401, 57.481, 157.512]
  Set speed (17.2 mm/s)
  Call Extruder(339.31730)
  MoveL 9241 to (505.89, 539.81, 164) mm, rotated rx 180 ry 0 rz 160 deg; joints [11.035, 54.83, -3.405, -142.417, 57.705, 157.647]
  Set speed (17.2 mm/s)
  Call Extruder(344.81529)
  MoveL 9242 to (504.22, 540.02, 164) mm, rotated rx 180 ry 0 rz 160 deg; joints [11.101, 54.554, -2.879, -142.441, 57.928, 157.79]
  Set speed (17.3 mm/s)
  Call Extruder(350.02835)
  MoveL 9243 to (502.63, 540.16, 164) mm, rotated rx 180 ry 0 rz 160 deg; joints [11.155, 54.291, -2.376, -142.473, 58.139, 157.93]
  Set speed (17.2 mm/s)
  Call Extruder(355.46519)
  MoveL 9244 to (500.97, 540.23, 164) mm, rotated rx -180 ry 0 rz 160 deg; joints [11.204, 54.015, -1.85, -142.513, 58.356, 158.081]
  Set speed (10.0 mm/s)
  MoveL 9245 to (500.97, 540.23, 168) mm, rotated rx 180 ry 0 rz 160 deg; joints [11.204, 53.464, -1.751, -142.342, 57.997, 157.757]
  Set speed (120.0 mm/s)
  MoveL 9246 to (499.37, 539.08, 168) mm, rotated rx 180 ry 0 rz 160 deg; joints [11.102, 53.157, -1.169, -142.559, 58.177, 158.013]
  Set speed (17.3 mm/s)
  Call Extruder(360.70802)
  MoveL 9247 to (497.76, 539.02, 168) mm, rotated rx -180 ry 0 rz 160 deg; joints [11.134, 52.887, -0.657, -142.615, 58.381, 158.168]
  Set speed (17.3 mm/s)
  Call Extruder(365.95137)
  MoveL 9248 to (496.15, 538.89, 168) mm, rotated rx -180 ry 0 rz 160 deg; joints [11.157, 52.616, -0.144, -142.679, 58.582, 158.327]
  Set speed (17.3 mm/s)
  Call Extruder(371.08765)
  MoveL 9249 to (494.59, 538.71, 168) mm, rotated rx -180 ry 0 rz 160 deg; joints [11.172, 52.352, 0.356, -142.75, 58.776, 158.486]
  Set speed (17.3 mm/s)
  Call Extruder(376.19238)
  MoveL 9250 to (493.04, 538.46, 168) mm, rotated rx 180 ry 0 rz 160 deg; joints [11.179, 52.091, 0.852, -142.828, 58.965, 158.648]
  Set speed (17.3 mm/s)
  Call Extruder(381.58116)
  MoveL 9251 to (491.42, 538.13, 168) mm, rotated rx 180 ry 0 rz 160 deg; joints [11.179, 51.816, 1.374, -142.918, 59.161, 158.821]
  Set speed (17.3 mm/s)
  Call Extruder(386.58565)
  MoveL 9252 to (489.93, 537.76, 168) mm, rotated rx -180 ry 0 rz 160 deg; joints [11.169, 51.562, 1.854, -143.009, 59.339, 158.986]
  Call Extruder(391.88257)
  MoveL 9253 to (488.36, 537.31, 168) mm, rotated rx -180 ry 0 rz 160 deg; joints [11.151, 51.296, 2.359, -143.113, 59.523, 159.162]
  Set speed (17.3 mm/s)
  Call Extruder(397.09588)
  MoveL 9254 to (486.84, 536.8, 168) mm, rotated rx 180 ry 0 rz 160 deg; joints [11.125, 51.036, 2.852, -143.224, 59.7, 159.338]
  Call Extruder(402.17687)
  MoveL 9255 to (485.38, 536.25, 168) mm, rotated rx -180 ry 0 rz 160 deg; joints [11.091, 50.785, 3.326, -143.339, 59.868, 159.512]
  Set speed (17.3 mm/s)
  Call Extruder(404.91253)
  MoveL 9256 to (484.61, 535.92, 168) mm, rotated rx 180 ry 0 rz 160 deg; joints [11.069, 50.652, 3.579, -143.404, 59.956, 159.606]
  Set speed (17.3 mm/s)
  Call Extruder(407.30807)
  MoveL 9257 to (483.93, 535.63, 168) mm, rotated rx 180 ry 0 rz 160 deg; joints [11.048, 50.536, 3.799, -143.462, 60.032, 159.689]
  Set speed (17.4 mm/s)
  Call Extruder(411.10425)
  MoveL 9258 to (482.87, 535.14, 168) mm, rotated rx 180 ry 0 rz 160 deg; joints [11.012, 50.353, 4.146, -143.557, 60.151, 159.821]
  Set speed (17.4 mm/s)
  Call Extruder(415.66595)
  MoveL 9259 to (481.63, 534.5, 168) mm, rotated rx -180 ry 0 rz 160 deg; joints [10.961, 50.136, 4.556, -143.678, 60.29, 159.981]
  Set speed (17.3 mm/s)
  Call Extruder(418.38959)
  MoveL 9260 to (480.89, 534.1, 168) mm, rotated rx 180 ry 0 rz 160 deg; joints [10.928, 50.009, 4.798, -143.753, 60.37, 160.076]
  Call Extruder(423.07820)
  MoveL 9261 to (479.65, 533.37, 168) mm, rotated rx -180 ry 0 rz 160 deg; joints [10.865, 49.792, 5.209, -143.886, 60.506, 160.241]
  Set speed (17.3 mm/s)
  Call Extruder(426.10594)
  MoveL 9262 to (478.86, 532.88, 168) mm, rotated rx 180 ry 0 rz 160 deg; joints [10.821, 49.654, 5.47, -143.974, 60.59, 160.348]
  Call Extruder(430.97803)
  MoveL 9263 to (477.62, 532.04, 168) mm, rotated rx -180 ry 0 rz 160 deg; joints [10.744, 49.435, 5.884, -144.122, 60.723, 160.521]
  Call Extruder(436.17619)
  MoveL 9264 to (476.33, 531.1, 168) mm, rotated rx -180 ry 0 rz 160 deg; joints [10.653, 49.208, 6.315, -144.287, 60.858, 160.705]
  Set speed (17.3 mm/s)
  Call Extruder(439.11597)
  MoveL 9265 to (475.62, 530.54, 168) mm, rotated rx -180 ry 0 rz 160 deg; joints [10.598, 49.082, 6.554, -144.383, 60.931, 160.809]
  Set speed (17.3 mm/s)
  Call Extruder(441.72482)
  MoveL 9266 to (475, 530.04, 168) mm, rotated rx 180 ry 0 rz 160 deg; joints [10.547, 48.971, 6.764, -144.47, 60.995, 160.901]
  Call Extruder(444.23982)
  MoveL 9267 to (474.4, 529.54, 168) mm, rotated rx -180 ry 0 rz 160 deg; joints [10.496, 48.866, 6.963, -144.555, 61.055, 160.99]
  Call Extruder(446.96880)
  MoveL 9268 to (473.78, 528.98, 168) mm, rotated rx 180 ry 0 rz 160 deg; joints [10.438, 48.753, 7.176, -144.649, 61.118, 161.087]
  Set speed (17.3 mm/s)
  Call Extruder(449.48871)
  MoveL 9269 to (473.21, 528.46, 168) mm, rotated rx -180 ry 0 rz 160 deg; joints [10.383, 48.651, 7.369, -144.738, 61.175, 161.176]
  Set speed (17.3 mm/s)
  Call Extruder(452.11252)
  MoveL 9270 to (472.63, 527.9, 168) mm, rotated rx -180 ry 0 rz 160 deg; joints [10.324, 48.546, 7.568, -144.832, 61.232, 161.269]
  Call Extruder(456.99100)
  MoveL 9271 to (471.58, 526.83, 168) mm, rotated rx -180 ry 0 rz 160 deg; joints [10.208, 48.356, 7.928, -145.01, 61.334, 161.44]
  Set speed (17.3 mm/s)
  Call Extruder(460.96115)
  MoveL 9272 to (470.75, 525.93, 168) mm, rotated rx -180 ry 0 rz 160 deg; joints [10.109, 48.206, 8.213, -145.16, 61.413, 161.579]
  Set speed (17.3 mm/s)
  Call Extruder(465.12755)
  MoveL 9273 to (469.92, 524.96, 168) mm, rotated rx -180 ry 0 rz 160 deg; joints [10, 48.053, 8.502, -145.32, 61.491, 161.724]
  Set speed (17.3 mm/s)
  Call Extruder(469.90496)
  MoveL 9274 to (469, 523.81, 168) mm, rotated rx -180 ry 0 rz 160 deg; joints [9.869, 47.883, 8.823, -145.508, 61.575, 161.889]
  Set speed (17.3 mm/s)
  Call Extruder(472.54400)
  MoveL 9275 to (468.52, 523.16, 168) mm, rotated rx 180 ry 0 rz 160 deg; joints [9.794, 47.792, 8.995, -145.614, 61.618, 161.98]
  Call Extruder(475.53009)
  MoveL 9276 to (467.98, 522.42, 168) mm, rotated rx 180 ry 0 rz 160 deg; joints [9.707, 47.692, 9.185, -145.735, 61.665, 162.082]
  Call Extruder(477.72224)
  MoveL 9277 to (467.6, 521.86, 168) mm, rotated rx -180 ry 0 rz 160 deg; joints [9.641, 47.62, 9.321, -145.826, 61.698, 162.157]
  Set speed (17.3 mm/s)
  Call Extruder(480.64657)
  MoveL 9278 to (467.11, 521.11, 168) mm, rotated rx 180 ry 0 rz 160 deg; joints [9.552, 47.526, 9.499, -145.947, 61.741, 162.256]
  Set speed (17.3 mm/s)
  Call Extruder(483.36612)
  MoveL 9279 to (466.66, 520.4, 168) mm, rotated rx -180 ry 0 rz 160 deg; joints [9.467, 47.441, 9.659, -146.062, 61.777, 162.347]
  Set speed (17.3 mm/s)
  Call Extruder(485.61357)
  MoveL 9280 to (466.31, 519.81, 168) mm, rotated rx -180 ry 0 rz 160 deg; joints [9.396, 47.373, 9.788, -146.157, 61.806, 162.422]
  Set speed (17.3 mm/s)
  Call Extruder(490.60364)
  MoveL 9281 to (465.56, 518.48, 168) mm, rotated rx -180 ry 0 rz 160 deg; joints [9.233, 47.227, 10.065, -146.372, 61.866, 162.588]
  Set speed (17.3 mm/s)
  Call Extruder(493.36076)
  MoveL 9282 to (465.16, 517.73, 168) mm, rotated rx -180 ry 0 rz 160 deg; joints [9.14, 47.15, 10.211, -146.493, 61.895, 162.678]
  Set speed (17.3 mm/s)
  Call Extruder(495.99313)
  MoveL 9283 to (464.81, 517, 168) mm, rotated rx -180 ry 0 rz 160 deg; joints [9.05, 47.079, 10.345, -146.609, 61.922, 162.763]
  Set speed (17.3 mm/s)
  Call Extruder(501.02836)
  MoveL 9284 to (464.16, 515.6, 168) mm, rotated rx 180 ry 0 rz 160 deg; joints [8.874, 46.949, 10.591, -146.833, 61.967, 162.925]
  Set speed (17.3 mm/s)
  Call Extruder(503.81470)
  MoveL 9285 to (463.83, 514.81, 168) mm, rotated rx 180 ry 0 rz 160 deg; joints [8.774, 46.881, 10.719, -146.959, 61.988, 163.013]
  Set speed (17.3 mm/s)
  Call Extruder(506.22723)
  MoveL 9286 to (463.56, 514.12, 168) mm, rotated rx 180 ry 0 rz 160 deg; joints [8.687, 46.825, 10.827, -147.069, 62.005, 163.089]
  Set speed (17.3 mm/s)
  Call Extruder(508.55962)
  MoveL 9287 to (463.3, 513.45, 168) mm, rotated rx -180 ry 0 rz 160 deg; joints [8.601, 46.771, 10.927, -147.175, 62.02, 163.162]
  Set speed (17.3 mm/s)
  Call Extruder(511.50663)
  MoveL 9288 to (463, 512.6, 168) mm, rotated rx 180 ry 0 rz 160 deg; joints [8.491, 46.707, 11.048, -147.311, 62.036, 163.253]
  Set speed (17.3 mm/s)
  Call Extruder(516.61644)
  MoveL 9289 to (462.52, 511.1, 168) mm, rotated rx -180 ry 0 rz 160 deg; joints [8.297, 46.603, 11.246, -147.547, 62.059, 163.408]
  Set speed (17.3 mm/s)
  Call Extruder(519.44861)
  MoveL 9290 to (462.29, 510.26, 168) mm, rotated rx 180 ry 0 rz 160 deg; joints [8.188, 46.55, 11.346, -147.68, 62.068, 163.492]
  Call Extruder(521.91318)
  MoveL 9291 to (462.1, 509.53, 168) mm, rotated rx 180 ry 0 rz 160 deg; joints [8.092, 46.506, 11.43, -147.795, 62.074, 163.565]
  Set speed (17.3 mm/s)
  Call Extruder(524.07278)
  MoveL 9292 to (461.94, 508.89, 168) mm, rotated rx -180 ry 0 rz 160 deg; joints [8.007, 46.469, 11.5, -147.897, 62.078, 163.628]
  Set speed (17.3 mm/s)
  Call Extruder(527.84239)
  MoveL 9293 to (461.69, 507.76, 168) mm, rotated rx 180 ry 0 rz 160 deg; joints [7.857, 46.409, 11.614, -148.074, 62.081, 163.736]
  Set speed (17.3 mm/s)
  Call Extruder(532.50133)
  MoveL 9294 to (461.44, 506.35, 168) mm, rotated rx -180 ry 0 rz 160 deg; joints [7.669, 46.342, 11.74, -148.295, 62.079, 163.867]
  Set speed (17.3 mm/s)
  Call Extruder(537.70833)
  MoveL 9295 to (461.2, 504.77, 168) mm, rotated rx 180 ry 0 rz 160 deg; joints [7.457, 46.276, 11.864, -148.543, 62.07, 164.011]
  Set speed (17.3 mm/s)
  Call Extruder(542.90487)
  MoveL 9296 to (461.04, 503.18, 168) mm, rotated rx -180 ry 0 rz 160 deg; joints [7.241, 46.222, 11.967, -148.79, 62.053, 164.149]
  Call Extruder(547.95019)
  MoveL 9297 to (460.95, 501.63, 168) mm, rotated rx 180 ry 0 rz 160 deg; joints [7.03, 46.179, 12.047, -149.031, 62.028, 164.279]
  Set speed (17.3 mm/s)
  Call Extruder(553.22689)
  MoveL 9298 to (460.91, 500.01, 168) mm, rotated rx 180 ry 0 rz 160 deg; joints [6.808, 46.144, 12.114, -149.282, 61.995, 164.411]
  Call Extruder(557.98253)
  MoveL 9299 to (460.94, 498.55, 168) mm, rotated rx -180 ry 0 rz 160 deg; joints [6.606, 46.123, 12.153, -149.507, 61.957, 164.525]
  Set speed (17.3 mm/s)
  Call Extruder(562.51784)
  MoveL 9300 to (461.02, 497.16, 168) mm, rotated rx 180 ry 0 rz 160 deg; joints [6.413, 46.111, 12.176, -149.721, 61.915, 164.63]
  Set speed (17.3 mm/s)
  Call Extruder(567.27484)
  MoveL 9301 to (461.15, 495.7, 168) mm, rotated rx -180 ry 0 rz 160 deg; joints [6.21, 46.107, 12.185, -149.944, 61.864, 164.737]
  Call Extruder(571.95145)
  MoveL 9302 to (461.34, 494.28, 168) mm, rotated rx 180 ry 0 rz 160 deg; joints [6.011, 46.112, 12.175, -150.161, 61.808, 164.838]
  Set speed (17.3 mm/s)
  Call Extruder(576.71738)
  MoveL 9303 to (461.58, 492.84, 168) mm, rotated rx 180 ry 0 rz 160 deg; joints [5.808, 46.125, 12.149, -150.38, 61.745, 164.936]
  Call Extruder(581.24726)
  MoveL 9304 to (461.86, 491.47, 168) mm, rotated rx 180 ry 0 rz 160 deg; joints [5.616, 46.147, 12.109, -150.585, 61.679, 165.025]
  Call Extruder(585.94135)
  MoveL 9305 to (462.2, 490.07, 168) mm, rotated rx 180 ry 0 rz 160 deg; joints [5.418, 46.177, 12.051, -150.795, 61.604, 165.113]
  Call Extruder(590.67607)
  MoveL 9306 to (462.59, 488.67, 168) mm, rotated rx 180 ry 0 rz 160 deg; joints [5.22, 46.217, 11.977, -151.004, 61.522, 165.197]
  Set speed (17.3 mm/s)
  Call Extruder(595.26573)
  MoveL 9307 to (463.03, 487.33, 168) mm, rotated rx 180 ry 0 rz 160 deg; joints [5.03, 46.264, 11.888, -151.203, 61.437, 165.274]
  Call Extruder(600.10295)
  MoveL 9308 to (463.53, 485.93, 168) mm, rotated rx -180 ry 0 rz 160 deg; joints [4.831, 46.321, 11.779, -151.408, 61.342, 165.351]
  Call Extruder(604.82166)
  MoveL 9309 to (464.08, 484.59, 168) mm, rotated rx -180 ry 0 rz 160 deg; joints [4.64, 46.386, 11.656, -151.604, 61.242, 165.421]
  Set speed (17.3 mm/s)
  Call Extruder(609.46388)
  MoveL 9310 to (464.67, 483.29, 168) mm, rotated rx -180 ry 0 rz 160 deg; joints [4.454, 46.459, 11.519, -151.792, 61.139, 165.485]
  Set speed (17.3 mm/s)
  Call Extruder(614.14954)
  MoveL 9311 to (465.31, 482, 168) mm, rotated rx 180 ry 0 rz 160 deg; joints [4.27, 46.54, 11.365, -151.977, 61.029, 165.544]
  Set speed (17.3 mm/s)
  Call Extruder(618.78599)
  MoveL 9312 to (465.99, 480.75, 168) mm, rotated rx -180 ry 0 rz 160 deg; joints [4.092, 46.628, 11.198, -152.154, 60.915, 165.598]
  Call Extruder(623.56115)
  MoveL 9313 to (466.73, 479.49, 168) mm, rotated rx 180 ry 0 rz 160 deg; joints [3.911, 46.727, 11.011, -152.331, 60.792, 165.648]
  Set speed (17.3 mm/s)
  Call Extruder(628.15321)
  MoveL 9314 to (467.5, 478.3, 168) mm, rotated rx 180 ry 0 rz 160 deg; joints [3.741, 46.83, 10.816, -152.496, 60.669, 165.692]
  Set speed (17.3 mm/s)
  Call Extruder(632.77335)
  MoveL 9315 to (468.31, 477.13, 168) mm, rotated rx -180 ry 0 rz 160 deg; joints [3.575, 46.941, 10.606, -152.655, 60.54, 165.73]
  Set speed (17.3 mm/s)
  Call Extruder(637.60142)
  MoveL 9316 to (469.2, 475.94, 168) mm, rotated rx 180 ry 0 rz 160 deg; joints [3.405, 47.065, 10.371, -152.816, 60.4, 165.765]
  Set speed (17.3 mm/s)
  Call Extruder(642.20416)
  MoveL 9317 to (470.09, 474.85, 168) mm, rotated rx -180 ry 0 rz 160 deg; joints [3.249, 47.191, 10.134, -152.961, 60.261, 165.793]
  Set speed (17.3 mm/s)
  Call Extruder(646.89040)
  MoveL 9318 to (471.03, 473.76, 168) mm, rotated rx 180 ry 0 rz 160 deg; joints [3.094, 47.326, 9.879, -153.103, 60.116, 165.816]
  Call Extruder(651.65568)
  MoveL 9319 to (472.04, 472.69, 168) mm, rotated rx -180 ry 0 rz 160 deg; joints [2.942, 47.47, 9.606, -153.24, 59.964, 165.834]
  Call Extruder(656.17915)
  MoveL 9320 to (473.02, 471.72, 168) mm, rotated rx 180 ry 0 rz 160 deg; joints [2.803, 47.613, 9.334, -153.362, 59.816, 165.846]
  Call Extruder(660.93694)
  MoveL 9321 to (474.1, 470.73, 168) mm, rotated rx -180 ry 0 rz 160 deg; joints [2.662, 47.771, 9.036, -153.483, 59.655, 165.852]
  Call Extruder(665.70355)
  MoveL 9322 to (475.21, 469.78, 168) mm, rotated rx -180 ry 0 rz 160 deg; joints [2.527, 47.936, 8.724, -153.596, 59.491, 165.853]
  Call Extruder(670.31093)
  MoveL 9323 to (476.33, 468.9, 168) mm, rotated rx -180 ry 0 rz 160 deg; joints [2.403, 48.101, 8.411, -153.698, 59.328, 165.848]
  Set speed (17.3 mm/s)
  Call Extruder(675.08208)
  MoveL 9324 to (477.51, 468.04, 168) mm, rotated rx 180 ry 0 rz 160 deg; joints [2.28, 48.278, 8.075, -153.795, 59.156, 165.838]
  Set speed (17.3 mm/s)
  Call Extruder(679.66981)
  MoveL 9325 to (478.67, 467.25, 168) mm, rotated rx -180 ry 0 rz 160 deg; joints [2.168, 48.455, 7.741, -153.879, 58.987, 165.822]
  Set speed (17.3 mm/s)
  Call Extruder(684.53259)
  MoveL 9326 to (479.94, 466.46, 168) mm, rotated rx -180 ry 0 rz 160 deg; joints [2.057, 48.647, 7.376, -153.96, 58.805, 165.798]
  Set speed (17.3 mm/s)
  Call Extruder(688.94848)
  MoveL 9327 to (481.12, 465.78, 168) mm, rotated rx 180 ry 0 rz 160 deg; joints [1.961, 48.827, 7.035, -154.025, 58.637, 165.772]
  Set speed (17.3 mm/s)
  Call Extruder(693.72475)
  MoveL 9328 to (482.41, 465.09, 168) mm, rotated rx 180 ry 0 rz 160 deg; joints [1.864, 49.027, 6.657, -154.088, 58.453, 165.738]
  Call Extruder(698.49024)
  MoveL 9329 to (483.74, 464.46, 168) mm, rotated rx 180 ry 0 rz 160 deg; joints [1.775, 49.232, 6.27, -154.14, 58.266, 165.698]
  Call Extruder(702.91293)
  MoveL 9330 to (484.98, 463.92, 168) mm, rotated rx -180 ry 0 rz 160 deg; joints [1.698, 49.426, 5.902, -154.181, 58.091, 165.655]
  Set speed (17.3 mm/s)
  Call Extruder(707.77540)
  MoveL 9331 to (486.37, 463.37, 168) mm, rotated rx -180 ry 0 rz 160 deg; joints [1.621, 49.643, 5.49, -154.217, 57.897, 165.602]
  Set speed (17.3 mm/s)
  Call Extruder(712.52581)
  MoveL 9332 to (487.75, 462.89, 168) mm, rotated rx -180 ry 0 rz 160 deg; joints [1.552, 49.86, 5.079, -154.242, 57.705, 165.544]
  Set speed (17.3 mm/s)
  Call Extruder(717.07247)
  MoveL 9333 to (489.08, 462.47, 168) mm, rotated rx 180 ry 0 rz 160 deg; joints [1.493, 50.072, 4.679, -154.257, 57.52, 165.483]
  Set speed (17.3 mm/s)
  Call Extruder(721.82588)
  MoveL 9334 to (490.49, 462.09, 168) mm, rotated rx 180 ry 0 rz 160 deg; joints [1.439, 50.296, 4.253, -154.264, 57.325, 165.413]
  Set speed (17.3 mm/s)
  Call Extruder(726.59314)
  MoveL 9335 to (491.92, 461.76, 168) mm, rotated rx -180 ry 0 rz 160 deg; joints [1.391, 50.525, 3.82, -154.262, 57.129, 165.337]
  Call Extruder(731.12731)
  MoveL 9336 to (493.29, 461.5, 168) mm, rotated rx -180 ry 0 rz 160 deg; joints [1.353, 50.745, 3.403, -154.25, 56.942, 165.259]
  Set speed (17.3 mm/s)
  Call Extruder(735.94064)
  MoveL 9337 to (494.75, 461.27, 168) mm, rotated rx -180 ry 0 rz 160 deg; joints [1.319, 50.982, 2.954, -154.229, 56.742, 165.17]
  Set speed (17.3 mm/s)
  Call Extruder(740.60189)
  MoveL 9338 to (496.17, 461.1, 168) mm, rotated rx -180 ry 0 rz 160 deg; joints [1.294, 51.213, 2.515, -154.199, 56.549, 165.078]
  Set speed (17.3 mm/s)
  Call Extruder(745.24902)
  MoveL 9339 to (497.59, 460.99, 168) mm, rotated rx 180 ry 0 rz 160 deg; joints [1.275, 51.446, 2.074, -154.16, 56.357, 164.981]
  Set speed (17.3 mm/s)
  Call Extruder(750.01790)
  MoveL 9340 to (499.05, 460.93, 168) mm, rotated rx 180 ry 0 rz 160 deg; joints [1.263, 51.687, 1.617, -154.112, 56.159, 164.876]
  Set speed (17.4 mm/s)
  Call Extruder(754.61029)
  MoveL 9341 to (500.47, 460.92, 168) mm, rotated rx -180 ry 0 rz 160 deg; joints [1.258, 51.921, 1.174, -154.056, 55.97, 164.769]
  Call Extruder(759.38382)
  MoveL 9342 to (501.93, 460.96, 168) mm, rotated rx -180 ry 0 rz 160 deg; joints [1.26, 52.165, 0.711, -153.989, 55.773, 164.652]
  Set speed (17.3 mm/s)
  Call Extruder(763.98483)
  MoveL 9343 to (503.35, 461.06, 168) mm, rotated rx 180 ry 0 rz 160 deg; joints [1.268, 52.402, 0.263, -153.916, 55.585, 164.535]
  Call Extruder(768.73844)
  MoveL 9344 to (504.8, 461.21, 168) mm, rotated rx 180 ry 0 rz 160 deg; joints [1.283, 52.646, -0.201, -153.832, 55.393, 164.407]
  Call Extruder(773.35537)
  MoveL 9345 to (506.2, 461.41, 168) mm, rotated rx 180 ry 0 rz 160 deg; joints [1.304, 52.884, -0.652, -153.742, 55.207, 164.279]
  Set speed (17.3 mm/s)
  Call Extruder(778.01589)
  MoveL 9346 to (507.61, 461.66, 168) mm, rotated rx 180 ry 0 rz 160 deg; joints [1.332, 53.125, -1.108, -153.643, 55.022, 164.144]
  Set speed (17.3 mm/s)
  Call Extruder(782.00006)
  MoveL 9347 to (508.81, 461.92, 168) mm, rotated rx -180 ry 0 rz 160 deg; joints [1.36, 53.33, -1.496, -153.552, 54.865, 164.025]
  Call Extruder(787.31764)
  MoveL 9348 to (510.39, 462.32, 168) mm, rotated rx -180 ry 0 rz 160 deg; joints [1.406, 53.603, -2.014, -153.422, 54.659, 163.86]
  Set speed (17.4 mm/s)
  Call Extruder(792.08547)
  MoveL 9349 to (511.8, 462.74, 168) mm, rotated rx 180 ry 0 rz 160 deg; joints [1.453, 53.847, -2.477, -153.296, 54.476, 163.707]
  Set speed (17.3 mm/s)
  Call Extruder(796.82965)
  MoveL 9350 to (513.18, 463.2, 168) mm, rotated rx -180 ry 0 rz 160 deg; joints [1.506, 54.088, -2.935, -153.163, 54.298, 163.551]
  Call Extruder(801.31634)
  MoveL 9351 to (514.47, 463.69, 168) mm, rotated rx 180 ry 0 rz 160 deg; joints [1.563, 54.315, -3.364, -153.031, 54.133, 163.399]
  Call Extruder(806.19875)
  MoveL 9352 to (515.85, 464.27, 168) mm, rotated rx 180 ry 0 rz 160 deg; joints [1.629, 54.56, -3.829, -152.879, 53.957, 163.229]
  Set speed (17.3 mm/s)
  Call Extruder(810.87016)
  MoveL 9353 to (517.16, 464.88, 168) mm, rotated rx -180 ry 0 rz 160 deg; joints [1.699, 54.792, -4.269, -152.727, 53.792, 163.062]
  Set speed (17.3 mm/s)
  Call Extruder(815.42740)
  MoveL 9354 to (518.4, 465.52, 168) mm, rotated rx -180 ry 0 rz 160 deg; joints [1.773, 55.015, -4.693, -152.572, 53.635, 162.896]
  Set speed (17.3 mm/s)
  Call Extruder(820.24759)
  MoveL 9355 to (519.7, 466.24, 168) mm, rotated rx 180 ry 0 rz 160 deg; joints [1.856, 55.249, -5.137, -152.402, 53.474, 162.717]
  Set speed (17.3 mm/s)
  Call Extruder(824.91801)
  MoveL 9356 to (520.92, 466.98, 168) mm, rotated rx 180 ry 0 rz 160 deg; joints [1.942, 55.473, -5.561, -152.231, 53.322, 162.54]
  Call Extruder(829.50126)
  MoveL 9357 to (522.1, 467.76, 168) mm, rotated rx -180 ry 0 rz 160 deg; joints [2.031, 55.688, -5.97, -152.057, 53.178, 162.364]
  Set speed (17.4 mm/s)
  Call Extruder(834.19434)
  MoveL 9358 to (523.27, 468.6, 168) mm, rotated rx 180 ry 0 rz 160 deg; joints [2.128, 55.906, -6.382, -151.873, 53.035, 162.18]
  Set speed (17.3 mm/s)
  Call Extruder(838.92647)
  MoveL 9359 to (524.42, 469.49, 168) mm, rotated rx 180 ry 0 rz 160 deg; joints [2.23, 56.121, -6.79, -151.683, 52.896, 161.993]
  Set speed (17.3 mm/s)
  Call Extruder(843.60141)
  MoveL 9360 to (525.53, 470.4, 168) mm, rotated rx -180 ry 0 rz 160 deg; joints [2.335, 56.329, -7.185, -151.49, 52.765, 161.806]
  Call Extruder(848.18054)
  MoveL 9361 to (526.58, 471.34, 168) mm, rotated rx 180 ry 0 rz 160 deg; joints [2.443, 56.528, -7.562, -151.296, 52.642, 161.62]
  Set speed (17.3 mm/s)
  Call Extruder(853.00047)
  MoveL 9362 to (527.65, 472.37, 168) mm, rotated rx -180 ry 0 rz 160 deg; joints [2.56, 56.733, -7.951, -151.088, 52.519, 161.423]
  Set speed (17.3 mm/s)
  Call Extruder(855.54519)
  MoveL 9363 to (528.19, 472.93, 168) mm, rotated rx 180 ry 0 rz 160 deg; joints [2.625, 56.838, -8.151, -150.976, 52.456, 161.319]
  Set speed (17.3 mm/s)
  Call Extruder(858.14012)
  MoveL 9364 to (528.74, 473.51, 168) mm, rotated rx 180 ry 0 rz 160 deg; joints [2.691, 56.944, -8.352, -150.861, 52.394, 161.212]
  Set speed (17.3 mm/s)
  Call Extruder(860.73408)
  MoveL 9365 to (529.27, 474.1, 168) mm, rotated rx 180 ry 0 rz 160 deg; joints [2.759, 57.049, -8.55, -150.745, 52.335, 161.105]
  Set speed (17.3 mm/s)
  Call Extruder(863.67216)
  MoveL 9366 to (529.86, 474.79, 168) mm, rotated rx -180 ry 0 rz 160 deg; joints [2.837, 57.165, -8.77, -150.612, 52.269, 160.984]
  Set speed (17.3 mm/s)
  Call Extruder(865.95754)
  MoveL 9367 to (530.31, 475.33, 168) mm, rotated rx -180 ry 0 rz 160 deg; joints [2.899, 57.253, -8.939, -150.508, 52.22, 160.889]
  Set speed (17.3 mm/s)
  Call Extruder(869.16169)
  MoveL 9368 to (530.92, 476.1, 168) mm, rotated rx -180 ry 0 rz 160 deg; joints [2.987, 57.375, -9.17, -150.361, 52.154, 160.756]
  Call Extruder(874.01715)
  MoveL 9369 to (531.81, 477.3, 168) mm, rotated rx -180 ry 0 rz 160 deg; joints [3.124, 57.554, -9.509, -150.135, 52.06, 160.555]
  Set speed (17.4 mm/s)
  Call Extruder(876.90166)
  MoveL 9370 to (532.32, 478.02, 168) mm, rotated rx -180 ry 0 rz 160 deg; joints [3.206, 57.657, -9.705, -150, 52.007, 160.435]
  Set speed (17.4 mm/s)
  Call Extruder(881.38861)
  MoveL 9371 to (533.08, 479.18, 168) mm, rotated rx 180 ry 0 rz 160 deg; joints [3.338, 57.812, -9.999, -149.788, 51.931, 160.249]
  Set speed (17.3 mm/s)
  Call Extruder(884.07102)
  MoveL 9372 to (533.51, 479.88, 168) mm, rotated rx 180 ry 0 rz 160 deg; joints [3.418, 57.902, -10.169, -149.66, 51.889, 160.139]
  Set speed (17.3 mm/s)
  Call Extruder(886.67532)
  MoveL 9373 to (533.91, 480.57, 168) mm, rotated rx -180 ry 0 rz 160 deg; joints [3.497, 57.986, -10.329, -149.536, 51.851, 160.032]
  Call Extruder(889.30177)
  MoveL 9374 to (534.31, 481.28, 168) mm, rotated rx -180 ry 0 rz 160 deg; joints [3.577, 58.07, -10.487, -149.41, 51.814, 159.924]
  Set speed (17.3 mm/s)
  Call Extruder(891.84712)
  MoveL 9375 to (534.68, 481.97, 168) mm, rotated rx 180 ry 0 rz 160 deg; joints [3.656, 58.148, -10.636, -149.288, 51.78, 159.821]
  Set speed (17.3 mm/s)
  Call Extruder(894.48808)
  MoveL 9376 to (535.04, 482.69, 168) mm, rotated rx 180 ry 0 rz 160 deg; joints [3.739, 58.227, -10.786, -149.161, 51.748, 159.713]
  Set speed (17.3 mm/s)
  Call Extruder(897.05560)
  MoveL 9377 to (535.38, 483.4, 168) mm, rotated rx 180 ry 0 rz 160 deg; joints [3.82, 58.301, -10.927, -149.037, 51.719, 159.61]
  Set speed (17.3 mm/s)
  Call Extruder(899.65544)
  MoveL 9378 to (535.72, 484.13, 168) mm, rotated rx -180 ry 0 rz 160 deg; joints [3.903, 58.374, -11.066, -148.911, 51.691, 159.505]
  Call Extruder(904.81667)
  MoveL 9379 to (536.33, 485.59, 168) mm, rotated rx 180 ry 0 rz 160 deg; joints [4.069, 58.512, -11.327, -148.662, 51.645, 159.3]
  Set speed (17.3 mm/s)
  Call Extruder(910.01881)
  MoveL 9380 to (536.89, 487.09, 168) mm, rotated rx 180 ry 0 rz 160 deg; joints [4.24, 58.641, -11.571, -148.41, 51.607, 159.097]
  Set speed (17.3 mm/s)
  Call Extruder(915.17857)
  MoveL 9381 to (537.38, 488.59, 168) mm, rotated rx -180 ry 0 rz 160 deg; joints [4.412, 58.758, -11.793, -148.162, 51.579, 158.899]
  Call Extruder(920.47910)
  MoveL 9382 to (537.82, 490.16, 168) mm, rotated rx 180 ry 0 rz 160 deg; joints [4.591, 58.867, -12.001, -147.907, 51.561, 158.7]
  Set speed (17.3 mm/s)
  Call Extruder(925.65572)
  MoveL 9383 to (538.2, 491.71, 168) mm, rotated rx -180 ry 0 rz 160 deg; joints [4.768, 58.964, -12.184, -147.66, 51.552, 158.51]
  Set speed (17.3 mm/s)
  Call Extruder(930.95314)
  MoveL 9384 to (538.51, 493.3, 168) mm, rotated rx -180 ry 0 rz 160 deg; joints [4.952, 59.051, -12.35, -147.409, 51.553, 158.321]
  Set speed (17.3 mm/s)
  Call Extruder(936.08254)
  MoveL 9385 to (538.75, 494.86, 168) mm, rotated rx 180 ry 0 rz 160 deg; joints [5.131, 59.125, -12.489, -147.168, 51.564, 158.144]
  Set speed (17.3 mm/s)
  Call Extruder(941.44796)
  MoveL 9386 to (538.93, 496.5, 168) mm, rotated rx 180 ry 0 rz 160 deg; joints [5.32, 59.189, -12.612, -146.92, 51.586, 157.965]
  Set speed (17.4 mm/s)
  Call Extruder(946.55896)
  MoveL 9387 to (539.04, 498.07, 168) mm, rotated rx -180 ry 0 rz 160 deg; joints [5.501, 59.24, -12.707, -146.686, 51.616, 157.8]
  Set speed (17.3 mm/s)
  Call Extruder(951.76262)
  MoveL 9388 to (539.08, 499.67, 168) mm, rotated rx 180 ry 0 rz 160 deg; joints [5.686, 59.279, -12.783, -146.452, 51.657, 157.639]
  Set speed (17.3 mm/s)
  Call Extruder(956.82227)
  MoveL 9389 to (539.07, 501.22, 168) mm, rotated rx 180 ry 0 rz 160 deg; joints [5.867, 59.307, -12.835, -146.228, 51.705, 157.49]
  Set speed (17.3 mm/s)
  Call Extruder(962.14840)
  MoveL 9390 to (538.98, 502.86, 168) mm, rotated rx 180 ry 0 rz 160 deg; joints [6.058, 59.323, -12.866, -145.997, 51.766, 157.34]
  Set speed (17.4 mm/s)
  Call Extruder(967.35524)
  MoveL 9391 to (538.83, 504.45, 168) mm, rotated rx -180 ry 0 rz 160 deg; joints [6.245, 59.328, -12.874, -145.776, 51.835, 157.202]
  Set speed (17.4 mm/s)
  Call Extruder(972.65439)
  MoveL 9392 to (538.61, 506.07, 168) mm, rotated rx -180 ry 0 rz 160 deg; joints [6.435, 59.32, -12.86, -145.556, 51.915, 157.069]
  Set speed (17.3 mm/s)
  Call Extruder(977.74962)
  MoveL 9393 to (538.34, 507.61, 168) mm, rotated rx -180 ry 0 rz 160 deg; joints [6.617, 59.301, -12.823, -145.351, 52, 156.95]
  Set speed (17.3 mm/s)
  Call Extruder(983.01352)
  MoveL 9394 to (537.99, 509.19, 168) mm, rotated rx 180 ry 0 rz 160 deg; joints [6.805, 59.269, -12.763, -145.144, 52.097, 156.836]
  Set speed (17.4 mm/s)
  Call Extruder(988.33530)
  MoveL 9395 to (537.57, 510.77, 168) mm, rotated rx -180 ry 0 rz 160 deg; joints [6.994, 59.225, -12.679, -144.941, 52.204, 156.73]
  Set speed (17.3 mm/s)
  Call Extruder(993.18671)
  MoveL 9396 to (537.13, 512.2, 168) mm, rotated rx 180 ry 0 rz 160 deg; joints [7.166, 59.174, -12.583, -144.763, 52.31, 156.641]
  Set speed (17.3 mm/s)
  Call Extruder(998.54269)
  MoveL 9397 to (536.59, 513.75, 168) mm, rotated rx -180 ry 0 rz 160 deg; joints [7.354, 59.106, -12.455, -144.572, 52.434, 156.552]
  Set speed (17.3 mm/s)
  Call Extruder(1003.79783)
  MoveL 9398 to (535.99, 515.25, 168) mm, rotated rx -180 ry 0 rz 160 deg; joints [7.537, 59.028, -12.306, -144.391, 52.564, 156.475]
  Set speed (17.4 mm/s)
  Call Extruder(1008.95826)
  MoveL 9399 to (535.34, 516.7, 168) mm, rotated rx 180 ry 0 rz 160 deg; joints [7.715, 58.941, -12.141, -144.22, 52.699, 156.407]
  Set speed (17.4 mm/s)
  Call Extruder(1014.19735)
  MoveL 9400 to (534.62, 518.14, 168) mm, rotated rx -180 ry 0 rz 160 deg; joints [7.894, 58.84, -11.949, -144.055, 52.844, 156.35]
  Set speed (17.3 mm/s)
  Call Extruder(1016.77398)
  MoveL 9401 to (534.25, 518.84, 168) mm, rotated rx -180 ry 0 rz 160 deg; joints [7.981, 58.786, -11.847, -143.977, 52.918, 156.325]
  Set speed (17.3 mm/s)
  Call Extruder(1019.38726)
  MoveL 9402 to (533.85, 519.54, 168) mm, rotated rx -180 ry 0 rz 160 deg; joints [8.069, 58.729, -11.739, -143.899, 52.994, 156.302]
  Set speed (17.3 mm/s)
  Call Extruder(1022.34352)
  MoveL 9403 to (533.39, 520.32, 168) mm, rotated rx 180 ry 0 rz 160 deg; joints [8.167, 58.662, -11.611, -143.813, 53.083, 156.279]
  Set speed (17.3 mm/s)
  Call Extruder(1025.00087)
  MoveL 9404 to (532.96, 521.01, 168) mm, rotated rx -180 ry 0 rz 160 deg; joints [8.256, 58.599, -11.491, -143.737, 53.164, 156.26]
  Set speed (17.3 mm/s)
  Call Extruder(1029.64275)
  MoveL 9405 to (532.17, 522.2, 168) mm, rotated rx 180 ry 0 rz 160 deg; joints [8.407, 58.481, -11.268, -143.61, 53.31, 156.235]
  Set speed (17.3 mm/s)
  Call Extruder(1032.41936)
  MoveL 9406 to (531.68, 522.9, 168) mm, rotated rx 180 ry 0 rz 160 deg; joints [8.497, 58.407, -11.128, -143.537, 53.4, 156.222]
  Set speed (17.3 mm/s)
  Call Extruder(1034.90380)
  MoveL 9407 to (531.23, 523.51, 168) mm, rotated rx -180 ry 0 rz 160 deg; joints [8.577, 58.339, -10.998, -143.473, 53.481, 156.214]
  Set speed (17.3 mm/s)
  Call Extruder(1037.57688)
  MoveL 9408 to (530.72, 524.16, 168) mm, rotated rx 180 ry 0 rz 160 deg; joints [8.661, 58.262, -10.853, -143.408, 53.571, 156.207]
  Set speed (17.3 mm/s)
  Call Extruder(1040.13324)
  MoveL 9409 to (530.23, 524.78, 168) mm, rotated rx 180 ry 0 rz 160 deg; joints [8.742, 58.187, -10.71, -143.346, 53.657, 156.203]
  Set speed (17.3 mm/s)
  Call Extruder(1042.84489)
  MoveL 9410 to (529.7, 525.41, 168) mm, rotated rx 180 ry 0 rz 160 deg; joints [8.826, 58.104, -10.553, -143.283, 53.75, 156.202]
  Set speed (17.3 mm/s)
  Call Extruder(1045.39656)
  MoveL 9411 to (529.18, 526, 168) mm, rotated rx 180 ry 0 rz 160 deg; joints [8.904, 58.025, -10.402, -143.225, 53.84, 156.202]
  Set speed (17.3 mm/s)
  Call Extruder(1048.44799)
  MoveL 9412 to (528.55, 526.7, 168) mm, rotated rx -180 ry 0 rz 160 deg; joints [8.997, 57.927, -10.216, -143.159, 53.947, 156.205]
  Set speed (17.4 mm/s)
  Call Extruder(1053.05022)
  MoveL 9413 to (527.56, 527.71, 168) mm, rotated rx 180 ry 0 rz 160 deg; joints [9.134, 57.772, -9.923, -143.064, 54.113, 156.217]
  Set speed (17.3 mm/s)
  Call Extruder(1055.79162)
  MoveL 9414 to (526.96, 528.3, 168) mm, rotated rx -180 ry 0 rz 160 deg; joints [9.214, 57.677, -9.743, -143.01, 54.214, 156.227]
  Call Extruder(1058.33401)
  MoveL 9415 to (526.39, 528.83, 168) mm, rotated rx 180 ry 0 rz 160 deg; joints [9.288, 57.587, -9.572, -142.963, 54.308, 156.239]
  Set speed (17.3 mm/s)
  Call Extruder(1061.37078)
  MoveL 9416 to (525.69, 529.46, 168) mm, rotated rx -180 ry 0 rz 160 deg; joints [9.374, 57.477, -9.363, -142.908, 54.422, 156.255]
  Set speed (17.3 mm/s)
  Call Extruder(1063.55178)
  MoveL 9417 to (525.18, 529.89, 168) mm, rotated rx -180 ry 0 rz 160 deg; joints [9.435, 57.396, -9.21, -142.87, 54.504, 156.269]
  Set speed (17.3 mm/s)
  Call Extruder(1066.72993)
  MoveL 9418 to (524.43, 530.51, 168) mm, rotated rx -180 ry 0 rz 160 deg; joints [9.523, 57.276, -8.982, -142.818, 54.625, 156.292]
  Set speed (17.3 mm/s)
  Call Extruder(1070.00936)
  MoveL 9419 to (523.64, 531.13, 168) mm, rotated rx -180 ry 0 rz 160 deg; joints [9.612, 57.149, -8.741, -142.767, 54.752, 156.319]
  Set speed (17.3 mm/s)
  Call Extruder(1074.00724)
  MoveL 9420 to (522.65, 531.86, 168) mm, rotated rx 180 ry 0 rz 160 deg; joints [9.717, 56.99, -8.44, -142.71, 54.907, 156.356]
  Set speed (17.3 mm/s)
  Call Extruder(1076.95159)
  MoveL 9421 to (521.9, 532.37, 168) mm, rotated rx 180 ry 0 rz 160 deg; joints [9.793, 56.871, -8.213, -142.671, 55.023, 156.387]
  Set speed (17.3 mm/s)
  Call Extruder(1079.16643)
  MoveL 9422 to (521.34, 532.75, 168) mm, rotated rx 180 ry 0 rz 160 deg; joints [9.849, 56.779, -8.04, -142.643, 55.111, 156.412]
  Call Extruder(1081.73668)
  MoveL 9423 to (520.67, 533.17, 168) mm, rotated rx -180 ry 0 rz 160 deg; joints [9.913, 56.672, -7.835, -142.612, 55.213, 156.442]
  Set speed (17.3 mm/s)
  Call Extruder(1084.32522)
  MoveL 9424 to (519.99, 533.59, 168) mm, rotated rx -180 ry 0 rz 160 deg; joints [9.976, 56.562, -7.627, -142.584, 55.317, 156.475]
  Set speed (17.3 mm/s)
  Call Extruder(1089.03132)
  MoveL 9425 to (518.74, 534.3, 168) mm, rotated rx -180 ry 0 rz 160 deg; joints [10.088, 56.358, -7.24, -142.536, 55.506, 156.54]
  Set speed (17.3 mm/s)
  Call Extruder(1092.20920)
  MoveL 9426 to (517.87, 534.76, 168) mm, rotated rx 180 ry 0 rz 160 deg; joints [10.16, 56.218, -6.974, -142.508, 55.635, 156.587]
  Set speed (17.3 mm/s)
  Call Extruder(1094.71919)
  MoveL 9427 to (517.18, 535.11, 168) mm, rotated rx -180 ry 0 rz 160 deg; joints [10.216, 56.105, -6.761, -142.488, 55.737, 156.626]
  Set speed (17.3 mm/s)
  Call Extruder(1097.38066)
  MoveL 9428 to (516.44, 535.46, 168) mm, rotated rx -180 ry 0 rz 160 deg; joints [10.273, 55.985, -6.532, -142.468, 55.846, 156.67]
  Set speed (17.3 mm/s)
  Call Extruder(1102.54182)
  MoveL 9429 to (514.99, 536.1, 168) mm, rotated rx -180 ry 0 rz 160 deg; joints [10.381, 55.747, -6.082, -142.437, 56.057, 156.76]
  Call Extruder(1107.65547)
  MoveL 9430 to (513.53, 536.67, 168) mm, rotated rx -180 ry 0 rz 160 deg; joints [10.482, 55.507, -5.626, -142.414, 56.267, 156.856]
  Set speed (17.3 mm/s)
  Call Extruder(1112.91241)
  MoveL 9431 to (512, 537.2, 168) mm, rotated rx 180 ry 0 rz 160 deg; joints [10.579, 55.256, -5.151, -142.397, 56.484, 156.961]
  Set speed (17.3 mm/s)
  Call Extruder(1117.71860)
  MoveL 9432 to (510.59, 537.63, 168) mm, rotated rx -180 ry 0 rz 160 deg; joints [10.663, 55.024, -4.709, -142.389, 56.682, 157.063]
  Set speed (17.3 mm/s)
  Call Extruder(1123.28588)
  MoveL 9433 to (508.93, 538.05, 168) mm, rotated rx -180 ry 0 rz 160 deg; joints [10.751, 54.75, -4.189, -142.39, 56.911, 157.189]
  Call Extruder(1128.66915)
  MoveL 9434 to (507.32, 538.39, 168) mm, rotated rx -180 ry 0 rz 160 deg; joints [10.83, 54.482, -3.682, -142.398, 57.132, 157.316]
  Set speed (17.3 mm/s)
  Call Extruder(1133.93396)
  MoveL 9435 to (505.72, 538.66, 168) mm, rotated rx 180 ry 0 rz 160 deg; joints [10.9, 54.217, -3.179, -142.414, 57.346, 157.447]
  Set speed (17.3 mm/s)
  Call Extruder(1138.96256)
  MoveL 9436 to (504.19, 538.86, 168) mm, rotated rx 180 ry 0 rz 160 deg; joints [10.96, 53.962, -2.696, -142.438, 57.55, 157.577]
  Call Extruder(1144.30987)
  MoveL 9437 to (502.56, 539, 168) mm, rotated rx -180 ry 0 rz 160 deg; joints [11.016, 53.69, -2.179, -142.471, 57.766, 157.72]
  Set speed (17.3 mm/s)
  Call Extruder(1149.55766)
  MoveL 9438 to (500.94, 539.07, 168) mm, rotated rx -180 ry 0 rz 160 deg; joints [11.063, 53.42, -1.669, -142.511, 57.975, 157.866]
  Call Extruder(1154.67985)
  MoveL 9439 to (499.37, 539.08, 168) mm, rotated rx 180 ry 0 rz 160 deg; joints [11.102, 53.157, -1.169, -142.559, 58.177, 158.013]
  Set speed (10.0 mm/s)
  MoveL 9440 to (499.37, 539.08, 172) mm, rotated rx 180 ry 0 rz 160 deg; joints [11.102, 52.609, -1.081, -142.383, 57.812, 157.683]
  Set speed (120.0 mm/s)
  MoveL 9441 to (499.41, 538.02, 172) mm, rotated rx -180 ry 0 rz 160 deg; joints [10.971, 52.582, -1.03, -142.536, 57.781, 157.776]
  Set speed (17.5 mm/s)
  Call Extruder(1159.84777)
  MoveL 9442 to (497.82, 537.97, 172) mm, rotated rx 180 ry 0 rz 160 deg; joints [11.002, 52.312, -0.522, -142.593, 57.982, 157.93]
  Set speed (17.5 mm/s)
  Call Extruder(1164.89614)
  MoveL 9443 to (496.26, 537.84, 172) mm, rotated rx 180 ry 0 rz 160 deg; joints [11.024, 52.049, -0.025, -142.657, 58.176, 158.083]
  Call Extruder(1169.84631)
  MoveL 9444 to (494.74, 537.67, 172) mm, rotated rx 180 ry 0 rz 160 deg; joints [11.039, 51.791, 0.461, -142.726, 58.363, 158.237]
  Set speed (17.5 mm/s)
  Call Extruder(1174.72492)
  MoveL 9445 to (493.24, 537.42, 172) mm, rotated rx -180 ry 0 rz 160 deg; joints [11.045, 51.537, 0.939, -142.803, 58.543, 158.393]
  Set speed (17.5 mm/s)
  Call Extruder(1179.67533)
  MoveL 9446 to (491.74, 537.12, 172) mm, rotated rx 180 ry 0 rz 160 deg; joints [11.044, 51.28, 1.421, -142.887, 58.723, 158.553]
  Call Extruder(1184.88436)
  MoveL 9447 to (490.17, 536.74, 172) mm, rotated rx -180 ry 0 rz 160 deg; joints [11.034, 51.012, 1.926, -142.984, 58.908, 158.726]
  Set speed (17.5 mm/s)
  Call Extruder(1190.59521)
  MoveL 9448 to (488.48, 536.25, 172) mm, rotated rx 180 ry 0 rz 160 deg; joints [11.014, 50.721, 2.474, -143.099, 59.106, 158.917]
  Set speed (17.5 mm/s)
  Call Extruder(1194.95529)
  MoveL 9449 to (487.2, 535.81, 172) mm, rotated rx 180 ry 0 rz 160 deg; joints [10.99, 50.501, 2.888, -143.194, 59.253, 159.066]
  Set speed (17.5 mm/s)
  Call Extruder(1197.85770)
  MoveL 9450 to (486.36, 535.5, 172) mm, rotated rx -180 ry 0 rz 160 deg; joints [10.971, 50.356, 3.162, -143.26, 59.349, 159.166]
  Set speed (17.5 mm/s)
  Call Extruder(1200.14057)
  MoveL 9451 to (485.7, 535.24, 172) mm, rotated rx 180 ry 0 rz 160 deg; joints [10.955, 50.242, 3.376, -143.314, 59.424, 159.245]
  Set speed (17.5 mm/s)
  Call Extruder(1205.38979)
  MoveL 9452 to (484.21, 534.6, 172) mm, rotated rx 180 ry 0 rz 160 deg; joints [10.91, 49.983, 3.863, -143.443, 59.591, 159.427]
  Call Extruder(1207.51050)
  MoveL 9453 to (483.61, 534.32, 172) mm, rotated rx -180 ry 0 rz 160 deg; joints [10.889, 49.879, 4.058, -143.497, 59.657, 159.502]
  Set speed (17.5 mm/s)
  Call Extruder(1210.00167)
  MoveL 9454 to (482.92, 533.98, 172) mm, rotated rx 180 ry 0 rz 160 deg; joints [10.862, 49.759, 4.285, -143.563, 59.733, 159.59]
  Set speed (17.5 mm/s)
  Call Extruder(1212.47659)
  MoveL 9455 to (482.24, 533.63, 172) mm, rotated rx 180 ry 0 rz 160 deg; joints [10.834, 49.64, 4.509, -143.63, 59.808, 159.677]
  Set speed (17.5 mm/s)
  Call Extruder(1215.06302)
  MoveL 9456 to (481.54, 533.24, 172) mm, rotated rx 180 ry 0 rz 160 deg; joints [10.802, 49.516, 4.741, -143.702, 59.884, 159.769]
  Set speed (17.5 mm/s)
  Call Extruder(1218.95845)
  MoveL 9457 to (480.49, 532.64, 172) mm, rotated rx -180 ry 0 rz 160 deg; joints [10.751, 49.333, 5.086, -143.813, 59.997, 159.907]
  Set speed (17.5 mm/s)
  Call Extruder(1222.97621)
  MoveL 9458 to (479.43, 531.99, 172) mm, rotated rx -180 ry 0 rz 160 deg; joints [10.692, 49.146, 5.436, -143.932, 60.109, 160.05]
  Set speed (17.5 mm/s)
  Call Extruder(1225.35322)
  MoveL 9459 to (478.82, 531.59, 172) mm, rotated rx -180 ry 0 rz 160 deg; joints [10.655, 49.038, 5.64, -144.005, 60.174, 160.135]
  Set speed (17.5 mm/s)
  Call Extruder(1230.52074)
  MoveL 9460 to (477.51, 530.67, 172) mm, rotated rx 180 ry 0 rz 160 deg; joints [10.568, 48.805, 6.077, -144.168, 60.31, 160.32]
  Set speed (17.5 mm/s)
  Call Extruder(1232.60759)
  MoveL 9461 to (476.99, 530.28, 172) mm, rotated rx 180 ry 0 rz 160 deg; joints [10.53, 48.713, 6.251, -144.236, 60.363, 160.395]
  Call Extruder(1235.16460)
  MoveL 9462 to (476.37, 529.79, 172) mm, rotated rx 180 ry 0 rz 160 deg; joints [10.482, 48.601, 6.46, -144.321, 60.426, 160.487]
  Set speed (17.5 mm/s)
  Call Extruder(1240.16133)
  MoveL 9463 to (475.17, 528.81, 172) mm, rotated rx 180 ry 0 rz 160 deg; joints [10.382, 48.387, 6.863, -144.491, 60.546, 160.666]
  Set speed (17.5 mm/s)
  Call Extruder(1242.70274)
  MoveL 9464 to (474.59, 528.29, 172) mm, rotated rx 180 ry 0 rz 160 deg; joints [10.328, 48.281, 7.063, -144.58, 60.605, 160.757]
  Set speed (17.5 mm/s)
  Call Extruder(1246.56572)
  MoveL 9465 to (473.7, 527.47, 172) mm, rotated rx 180 ry 0 rz 160 deg; joints [10.243, 48.121, 7.362, -144.718, 60.691, 160.896]
  Set speed (17.5 mm/s)
  Call Extruder(1250.63460)
  MoveL 9466 to (472.81, 526.59, 172) mm, rotated rx 180 ry 0 rz 160 deg; joints [10.147, 47.958, 7.669, -144.868, 60.777, 161.041]
  Set speed (17.5 mm/s)
  Call Extruder(1253.10771)
  MoveL 9467 to (472.28, 526.03, 172) mm, rotated rx -180 ry 0 rz 160 deg; joints [10.087, 47.861, 7.851, -144.961, 60.827, 161.129]
  Set speed (17.5 mm/s)
  Call Extruder(1255.21360)
  MoveL 9468 to (471.84, 525.55, 172) mm, rotated rx 180 ry 0 rz 160 deg; joints [10.034, 47.78, 8.003, -145.041, 60.868, 161.204]
  Set speed (17.5 mm/s)
  Call Extruder(1257.72980)
  MoveL 9469 to (471.32, 524.97, 172) mm, rotated rx 180 ry 0 rz 160 deg; joints [9.969, 47.685, 8.183, -145.138, 60.916, 161.293]
  Set speed (17.5 mm/s)
  Call Extruder(1260.19823)
  MoveL 9470 to (470.82, 524.39, 172) mm, rotated rx -180 ry 0 rz 160 deg; joints [9.904, 47.593, 8.355, -145.234, 60.962, 161.38]
  Set speed (17.5 mm/s)
  Call Extruder(1262.74971)
  MoveL 9471 to (470.32, 523.78, 172) mm, rotated rx 180 ry 0 rz 160 deg; joints [9.834, 47.499, 8.531, -145.335, 61.007, 161.47]
  Set speed (17.5 mm/s)
  Call Extruder(1265.47564)
  MoveL 9472 to (469.8, 523.12, 172) mm, rotated rx -180 ry 0 rz 160 deg; joints [9.758, 47.402, 8.714, -145.445, 61.053, 161.565]
  Set speed (17.5 mm/s)
  Call Extruder(1270.49699)
  MoveL 9473 to (468.88, 521.86, 172) mm, rotated rx 180 ry 0 rz 160 deg; joints [9.612, 47.229, 9.039, -145.651, 61.132, 161.74]
  Set speed (17.5 mm/s)
  Call Extruder(1275.33439)
  MoveL 9474 to (468.05, 520.62, 172) mm, rotated rx -180 ry 0 rz 160 deg; joints [9.465, 47.069, 9.339, -145.853, 61.202, 161.907]
  Set speed (17.5 mm/s)
  Call Extruder(1277.77266)
  MoveL 9475 to (467.65, 519.98, 172) mm, rotated rx -180 ry 0 rz 160 deg; joints [9.389, 46.992, 9.484, -145.957, 61.235, 161.99]
  Set speed (17.5 mm/s)
  Call Extruder(1280.54108)
  MoveL 9476 to (467.2, 519.25, 172) mm, rotated rx 180 ry 0 rz 160 deg; joints [9.3, 46.906, 9.645, -146.076, 61.27, 162.084]
  Set speed (17.5 mm/s)
  Call Extruder(1285.43431)
  MoveL 9477 to (466.46, 517.93, 172) mm, rotated rx 180 ry 0 rz 160 deg; joints [9.139, 46.76, 9.918, -146.29, 61.327, 162.249]
  Set speed (17.5 mm/s)
  Call Extruder(1290.11121)
  MoveL 9478 to (465.8, 516.64, 172) mm, rotated rx -180 ry 0 rz 160 deg; joints [8.98, 46.629, 10.163, -146.497, 61.374, 162.404]
  Call Extruder(1295.32125)
  MoveL 9479 to (465.13, 515.17, 172) mm, rotated rx 180 ry 0 rz 160 deg; joints [8.797, 46.493, 10.42, -146.733, 61.419, 162.575]
  Set speed (17.5 mm/s)
  Call Extruder(1298.30705)
  MoveL 9480 to (464.77, 514.32, 172) mm, rotated rx 180 ry 0 rz 160 deg; joints [8.689, 46.419, 10.558, -146.869, 61.441, 162.671]
  Call Extruder(1300.71606)
  MoveL 9481 to (464.5, 513.63, 172) mm, rotated rx 180 ry 0 rz 160 deg; joints [8.601, 46.362, 10.666, -146.979, 61.457, 162.748]
  Set speed (17.5 mm/s)
  Call Extruder(1305.52495)
  MoveL 9482 to (463.99, 512.23, 172) mm, rotated rx -180 ry 0 rz 160 deg; joints [8.421, 46.253, 10.869, -147.203, 61.483, 162.9]
  Set speed (17.5 mm/s)
  Call Extruder(1310.38686)
  MoveL 9483 to (463.54, 510.79, 172) mm, rotated rx -180 ry 0 rz 160 deg; joints [8.236, 46.153, 11.057, -147.43, 61.503, 163.05]
  Set speed (17.5 mm/s)
  Call Extruder(1315.57568)
  MoveL 9484 to (463.11, 509.25, 172) mm, rotated rx -180 ry 0 rz 160 deg; joints [8.033, 46.056, 11.24, -147.676, 61.516, 163.207]
  Set speed (17.5 mm/s)
  Call Extruder(1319.79247)
  MoveL 9485 to (462.82, 507.97, 172) mm, rotated rx -180 ry 0 rz 160 deg; joints [7.866, 45.985, 11.373, -147.876, 61.52, 163.332]
  Set speed (17.5 mm/s)
  Call Extruder(1325.69669)
  MoveL 9486 to (462.48, 506.18, 172) mm, rotated rx 180 ry 0 rz 160 deg; joints [7.627, 45.897, 11.538, -148.159, 61.517, 163.503]
  Set speed (17.5 mm/s)
  Call Extruder(1330.72567)
  MoveL 9487 to (462.26, 504.64, 172) mm, rotated rx -180 ry 0 rz 160 deg; joints [7.42, 45.833, 11.657, -148.4, 61.506, 163.644]
  Set speed (17.5 mm/s)
  Call Extruder(1335.74206)
  MoveL 9488 to (462.1, 503.1, 172) mm, rotated rx 180 ry 0 rz 160 deg; joints [7.211, 45.779, 11.758, -148.642, 61.488, 163.78]
  Set speed (17.5 mm/s)
  Call Extruder(1340.91113)
  MoveL 9489 to (462, 501.5, 172) mm, rotated rx 180 ry 0 rz 160 deg; joints [6.994, 45.735, 11.841, -148.89, 61.46, 163.917]
  Set speed (17.5 mm/s)
  Call Extruder(1345.58690)
  MoveL 9490 to (461.97, 500.05, 172) mm, rotated rx 180 ry 0 rz 160 deg; joints [6.796, 45.705, 11.898, -149.115, 61.429, 164.036]
  Set speed (17.5 mm/s)
  Call Extruder(1350.30215)
  MoveL 9491 to (462, 498.59, 172) mm, rotated rx 180 ry 0 rz 160 deg; joints [6.595, 45.683, 11.939, -149.34, 61.39, 164.153]
  Set speed (17.5 mm/s)
  Call Extruder(1354.74715)
  MoveL 9492 to (462.07, 497.22, 172) mm, rotated rx 180 ry 0 rz 160 deg; joints [6.404, 45.67, 11.963, -149.552, 61.348, 164.259]
  Set speed (17.5 mm/s)
  Call Extruder(1359.26488)
  MoveL 9493 to (462.2, 495.82, 172) mm, rotated rx 180 ry 0 rz 160 deg; joints [6.211, 45.666, 11.97, -149.765, 61.298, 164.363]
  Set speed (17.5 mm/s)
  Call Extruder(1363.78664)
  MoveL 9494 to (462.38, 494.44, 172) mm, rotated rx 180 ry 0 rz 160 deg; joints [6.017, 45.671, 11.961, -149.977, 61.243, 164.463]
  Call Extruder(1368.39158)
  MoveL 9495 to (462.62, 493.03, 172) mm, rotated rx -180 ry 0 rz 160 deg; joints [5.82, 45.684, 11.936, -150.19, 61.18, 164.56]
  Set speed (17.5 mm/s)
  Call Extruder(1372.82845)
  MoveL 9496 to (462.89, 491.68, 172) mm, rotated rx -180 ry 0 rz 160 deg; joints [5.631, 45.706, 11.896, -150.393, 61.114, 164.65]
  Call Extruder(1377.28485)
  MoveL 9497 to (463.22, 490.34, 172) mm, rotated rx -180 ry 0 rz 160 deg; joints [5.442, 45.735, 11.841, -150.594, 61.041, 164.736]
  Call Extruder(1381.80205)
  MoveL 9498 to (463.6, 489, 172) mm, rotated rx 180 ry 0 rz 160 deg; joints [5.252, 45.774, 11.769, -150.795, 60.962, 164.819]
  Set speed (17.5 mm/s)
  Call Extruder(1386.40036)
  MoveL 9499 to (464.04, 487.64, 172) mm, rotated rx 180 ry 0 rz 160 deg; joints [5.06, 45.821, 11.68, -150.996, 60.876, 164.899]
  Set speed (17.5 mm/s)
  Call Extruder(1390.92448)
  MoveL 9500 to (464.52, 486.33, 172) mm, rotated rx -180 ry 0 rz 160 deg; joints [4.874, 45.876, 11.576, -151.189, 60.785, 164.973]
  Set speed (17.5 mm/s)
  Call Extruder(1394.63711)
  MoveL 9501 to (464.94, 485.26, 172) mm, rotated rx -180 ry 0 rz 160 deg; joints [4.722, 45.927, 11.482, -151.345, 60.707, 165.031]
  Set speed (17.5 mm/s)
  Call Extruder(1400.00021)
  MoveL 9502 to (465.62, 483.74, 172) mm, rotated rx -180 ry 0 rz 160 deg; joints [4.506, 46.011, 11.323, -151.564, 60.586, 165.107]
  Set speed (17.5 mm/s)
  Call Extruder(1404.44722)
  MoveL 9503 to (466.23, 482.51, 172) mm, rotated rx 180 ry 0 rz 160 deg; joints [4.331, 46.09, 11.176, -151.74, 60.481, 165.166]
  Call Extruder(1409.00509)
  MoveL 9504 to (466.91, 481.27, 172) mm, rotated rx 180 ry 0 rz 160 deg; joints [4.154, 46.178, 11.01, -151.916, 60.367, 165.221]
  Set speed (17.5 mm/s)
  Call Extruder(1413.62531)
  MoveL 9505 to (467.63, 480.04, 172) mm, rotated rx 180 ry 0 rz 160 deg; joints [3.978, 46.275, 10.828, -152.089, 60.247, 165.272]
  Set speed (17.5 mm/s)
  Call Extruder(1418.06470)
  MoveL 9506 to (468.37, 478.88, 172) mm, rotated rx 180 ry 0 rz 160 deg; joints [3.813, 46.376, 10.639, -152.249, 60.127, 165.316]
  Set speed (17.5 mm/s)
  Call Extruder(1422.57850)
  MoveL 9507 to (469.17, 477.73, 172) mm, rotated rx 180 ry 0 rz 160 deg; joints [3.65, 46.487, 10.431, -152.406, 60, 165.355]
  Set speed (17.5 mm/s)
  Call Extruder(1427.18853)
  MoveL 9508 to (470.03, 476.59, 172) mm, rotated rx -180 ry 0 rz 160 deg; joints [3.487, 46.607, 10.206, -152.56, 59.866, 165.39]
  Set speed (17.5 mm/s)
  Call Extruder(1431.56619)
  MoveL 9509 to (470.88, 475.54, 172) mm, rotated rx -180 ry 0 rz 160 deg; joints [3.337, 46.728, 9.978, -152.7, 59.734, 165.418]
  Set speed (17.5 mm/s)
  Call Extruder(1436.15585)
  MoveL 9510 to (471.82, 474.47, 172) mm, rotated rx -180 ry 0 rz 160 deg; joints [3.184, 46.862, 9.727, -152.839, 59.591, 165.442]
  Set speed (17.5 mm/s)
  Call Extruder(1440.75100)
  MoveL 9511 to (472.79, 473.43, 172) mm, rotated rx -180 ry 0 rz 160 deg; joints [3.037, 47.004, 9.461, -152.972, 59.443, 165.46]
  Set speed (17.5 mm/s)
  Call Extruder(1445.08971)
  MoveL 9512 to (473.75, 472.49, 172) mm, rotated rx 180 ry 0 rz 160 deg; joints [2.902, 47.144, 9.198, -153.09, 59.3, 165.473]
  Set speed (17.5 mm/s)
  Call Extruder(1449.76429)
  MoveL 9513 to (474.81, 471.51, 172) mm, rotated rx 180 ry 0 rz 160 deg; joints [2.763, 47.301, 8.903, -153.209, 59.142, 165.48]
  Set speed (17.5 mm/s)
  Call Extruder(1454.17496)
  MoveL 9514 to (475.85, 470.63, 172) mm, rotated rx -180 ry 0 rz 160 deg; joints [2.637, 47.456, 8.612, -153.315, 58.989, 165.482]
  Set speed (17.5 mm/s)
  Call Extruder(1458.61800)
  MoveL 9515 to (476.93, 469.77, 172) mm, rotated rx 180 ry 0 rz 160 deg; joints [2.516, 47.618, 8.309, -153.414, 58.832, 165.479]
  Set speed (17.4 mm/s)
  Call Extruder(1461.03321)
  MoveL 9516 to (477.52, 469.32, 172) mm, rotated rx 180 ry 0 rz 160 deg; joints [2.452, 47.707, 8.141, -153.465, 58.746, 165.475]
  Set speed (17.4 mm/s)
  Call Extruder(1463.15933)
  MoveL 9517 to (478.06, 468.94, 172) mm, rotated rx -180 ry 0 rz 160 deg; joints [2.398, 47.788, 7.988, -153.506, 58.668, 165.469]
  Set speed (17.5 mm/s)
  Call Extruder(1467.85164)
  MoveL 9518 to (479.26, 468.12, 172) mm, rotated rx 180 ry 0 rz 160 deg; joints [2.283, 47.971, 7.644, -153.594, 58.495, 165.454]
  Set speed (17.5 mm/s)
  Call Extruder(1472.41525)
  MoveL 9519 to (480.46, 467.38, 172) mm, rotated rx -180 ry 0 rz 160 deg; joints [2.177, 48.155, 7.299, -153.67, 58.324, 165.433]
  Call Extruder(1476.94368)
  MoveL 9520 to (481.67, 466.68, 172) mm, rotated rx -180 ry 0 rz 160 deg; joints [2.078, 48.343, 6.946, -153.737, 58.151, 165.406]
  Set speed (17.5 mm/s)
  Call Extruder(1482.42813)
  MoveL 9521 to (483.18, 465.9, 172) mm, rotated rx -180 ry 0 rz 160 deg; joints [1.967, 48.576, 6.508, -153.807, 57.939, 165.366]
  Set speed (17.4 mm/s)
  Call Extruder(1486.00153)
  MoveL 9522 to (484.18, 465.42, 172) mm, rotated rx -180 ry 0 rz 160 deg; joints [1.9, 48.732, 6.214, -153.846, 57.799, 165.335]
  Set speed (17.5 mm/s)
  Call Extruder(1490.54163)
  MoveL 9523 to (485.46, 464.86, 172) mm, rotated rx 180 ry 0 rz 160 deg; joints [1.82, 48.934, 5.835, -153.888, 57.619, 165.291]
  Call Extruder(1494.90004)
  MoveL 9524 to (486.72, 464.37, 172) mm, rotated rx -180 ry 0 rz 160 deg; joints [1.75, 49.133, 5.462, -153.919, 57.445, 165.243]
  Set speed (17.5 mm/s)
  Call Extruder(1499.56870)
  MoveL 9525 to (488.08, 463.89, 172) mm, rotated rx 180 ry 0 rz 160 deg; joints [1.682, 49.349, 5.055, -153.943, 57.256, 165.186]
  Set speed (17.5 mm/s)
  Call Extruder(1503.93952)
  MoveL 9526 to (489.37, 463.49, 172) mm, rotated rx 180 ry 0 rz 160 deg; joints [1.625, 49.555, 4.667, -153.958, 57.078, 165.127]
  Set speed (17.5 mm/s)
  Call Extruder(1508.62651)
  MoveL 9527 to (490.77, 463.11, 172) mm, rotated rx 180 ry 0 rz 160 deg; joints [1.57, 49.78, 4.244, -153.964, 56.887, 165.058]
  Set speed (17.5 mm/s)
  Call Extruder(1512.95141)
  MoveL 9528 to (492.08, 462.81, 172) mm, rotated rx 180 ry 0 rz 160 deg; joints [1.527, 49.991, 3.848, -153.961, 56.709, 164.988]
  Set speed (17.5 mm/s)
  Call Extruder(1517.50366)
  MoveL 9529 to (493.46, 462.54, 172) mm, rotated rx -180 ry 0 rz 160 deg; joints [1.487, 50.215, 3.426, -153.95, 56.521, 164.909]
  Set speed (17.5 mm/s)
  Call Extruder(1522.12821)
  MoveL 9530 to (494.88, 462.32, 172) mm, rotated rx -180 ry 0 rz 160 deg; joints [1.454, 50.446, 2.992, -153.929, 56.329, 164.823]
  Set speed (17.5 mm/s)
  Call Extruder(1526.72520)
  MoveL 9531 to (496.29, 462.16, 172) mm, rotated rx -180 ry 0 rz 160 deg; joints [1.429, 50.678, 2.556, -153.898, 56.139, 164.731]
  Set speed (17.5 mm/s)
  Call Extruder(1531.09051)
  MoveL 9532 to (497.64, 462.05, 172) mm, rotated rx 180 ry 0 rz 160 deg; joints [1.41, 50.9, 2.138, -153.862, 55.958, 164.639]
  Set speed (17.5 mm/s)
  Call Extruder(1535.75732)
  MoveL 9533 to (499.08, 461.98, 172) mm, rotated rx 180 ry 0 rz 160 deg; joints [1.398, 51.139, 1.688, -153.813, 55.766, 164.535]
  Set speed (17.5 mm/s)
  Call Extruder(1540.19188)
  MoveL 9534 to (500.45, 461.98, 172) mm, rotated rx 180 ry 0 rz 160 deg; joints [1.393, 51.368, 1.257, -153.758, 55.583, 164.431]
  Set speed (17.5 mm/s)
  Call Extruder(1544.79471)
  MoveL 9535 to (501.88, 462.02, 172) mm, rotated rx 180 ry 0 rz 160 deg; joints [1.394, 51.607, 0.807, -153.693, 55.394, 164.317]
  Set speed (17.5 mm/s)
  Call Extruder(1549.24900)
  MoveL 9536 to (503.26, 462.11, 172) mm, rotated rx -180 ry 0 rz 160 deg; joints [1.401, 51.839, 0.37, -153.621, 55.213, 164.201]
  Set speed (17.5 mm/s)
  Call Extruder(1553.83811)
  MoveL 9537 to (504.67, 462.26, 172) mm, rotated rx 180 ry 0 rz 160 deg; joints [1.416, 52.078, -0.081, -153.539, 55.027, 164.077]
  Set speed (17.5 mm/s)
  Call Extruder(1558.26452)
  MoveL 9538 to (506.03, 462.45, 172) mm, rotated rx 180 ry 0 rz 160 deg; joints [1.435, 52.309, -0.516, -153.451, 54.85, 163.952]
  Set speed (17.5 mm/s)
  Call Extruder(1562.87183)
  MoveL 9539 to (507.43, 462.71, 172) mm, rotated rx 180 ry 0 rz 160 deg; joints [1.463, 52.55, -0.969, -153.352, 54.667, 163.817]
  Set speed (17.5 mm/s)
  Call Extruder(1567.33738)
  MoveL 9540 to (508.78, 463, 172) mm, rotated rx -180 ry 0 rz 160 deg; joints [1.495, 52.783, -1.408, -153.248, 54.492, 163.681]
  Set speed (17.5 mm/s)
  Call Extruder(1571.83705)
  MoveL 9541 to (510.13, 463.35, 172) mm, rotated rx -180 ry 0 rz 160 deg; joints [1.534, 53.017, -1.849, -153.135, 54.319, 163.54]
  Call Extruder(0.00000)
  Call Extruder(4.53732)
  MoveL 9542 to (511.48, 463.75, 172) mm, rotated rx 180 ry 0 rz 160 deg; joints [1.579, 53.252, -2.292, -153.014, 54.146, 163.393]
  Set speed (17.5 mm/s)
  Call Extruder(9.12932)
  MoveL 9543 to (512.82, 464.2, 172) mm, rotated rx -180 ry 0 rz 160 deg; joints [1.631, 53.488, -2.738, -152.884, 53.975, 163.239]
  Set speed (17.5 mm/s)
  Call Extruder(13.56147)
  MoveL 9544 to (514.11, 464.69, 172) mm, rotated rx 180 ry 0 rz 160 deg; joints [1.686, 53.715, -3.166, -152.751, 53.812, 163.087]
  Set speed (17.5 mm/s)
  Call Extruder(18.15913)
  MoveL 9545 to (515.42, 465.24, 172) mm, rotated rx -180 ry 0 rz 160 deg; joints [1.75, 53.949, -3.605, -152.607, 53.647, 162.925]
  Call Extruder(22.70021)
  MoveL 9546 to (516.69, 465.83, 172) mm, rotated rx 180 ry 0 rz 160 deg; joints [1.818, 54.177, -4.036, -152.457, 53.488, 162.761]
  Set speed (17.5 mm/s)
  Call Extruder(27.03937)
  MoveL 9547 to (517.89, 466.44, 172) mm, rotated rx 180 ry 0 rz 160 deg; joints [1.888, 54.393, -4.443, -152.308, 53.34, 162.601]
  Set speed (17.5 mm/s)
  Call Extruder(31.73684)
  MoveL 9548 to (519.16, 467.15, 172) mm, rotated rx -180 ry 0 rz 160 deg; joints [1.97, 54.623, -4.878, -152.14, 53.183, 162.424]
  Call Extruder(36.16803)
  MoveL 9549 to (520.33, 467.86, 172) mm, rotated rx -180 ry 0 rz 160 deg; joints [2.051, 54.838, -5.283, -151.975, 53.04, 162.254]
  Set speed (17.5 mm/s)
  Call Extruder(40.77683)
  MoveL 9550 to (521.52, 468.65, 172) mm, rotated rx -180 ry 0 rz 160 deg; joints [2.142, 55.058, -5.696, -151.798, 52.896, 162.074]
  Call Extruder(45.20483)
  MoveL 9551 to (522.64, 469.45, 172) mm, rotated rx 180 ry 0 rz 160 deg; joints [2.233, 55.265, -6.088, -151.623, 52.763, 161.899]
  Set speed (17.5 mm/s)
  Call Extruder(49.73230)
  MoveL 9552 to (523.75, 470.3, 172) mm, rotated rx 180 ry 0 rz 160 deg; joints [2.332, 55.473, -6.48, -151.439, 52.631, 161.717]
  Set speed (17.5 mm/s)
  Call Extruder(54.10125)
  MoveL 9553 to (524.79, 471.17, 172) mm, rotated rx 180 ry 0 rz 160 deg; joints [2.431, 55.67, -6.851, -151.256, 52.509, 161.54]
  Call Extruder(58.84673)
  MoveL 9554 to (525.89, 472.14, 172) mm, rotated rx -180 ry 0 rz 160 deg; joints [2.543, 55.879, -7.245, -151.054, 52.383, 161.346]
  Call Extruder(63.66298)
  MoveL 9555 to (526.96, 473.18, 172) mm, rotated rx 180 ry 0 rz 160 deg; joints [2.662, 56.085, -7.634, -150.843, 52.261, 161.147]
  Set speed (17.5 mm/s)
  Call Extruder(68.22710)
  MoveL 9556 to (527.94, 474.2, 172) mm, rotated rx -180 ry 0 rz 160 deg; joints [2.778, 56.275, -7.993, -150.639, 52.153, 160.957]
  Call Extruder(70.93938)
  MoveL 9557 to (528.5, 474.83, 172) mm, rotated rx 180 ry 0 rz 160 deg; joints [2.85, 56.385, -8.2, -150.516, 52.091, 160.844]
  Set speed (17.5 mm/s)
  Call Extruder(73.33043)
  MoveL 9558 to (528.98, 475.39, 172) mm, rotated rx -180 ry 0 rz 160 deg; joints [2.914, 56.48, -8.38, -150.407, 52.038, 160.744]
  Set speed (17.5 mm/s)
  Call Extruder(75.93278)
  MoveL 9559 to (529.5, 476, 172) mm, rotated rx -180 ry 0 rz 160 deg; joints [2.985, 56.583, -8.573, -150.288, 51.983, 160.635]
  Call Extruder(78.55721)
  MoveL 9560 to (530.01, 476.64, 172) mm, rotated rx -180 ry 0 rz 160 deg; joints [3.057, 56.684, -8.764, -150.166, 51.929, 160.524]
  Set speed (17.5 mm/s)
  Call Extruder(83.48359)
  MoveL 9561 to (530.92, 477.86, 172) mm, rotated rx 180 ry 0 rz 160 deg; joints [3.197, 56.867, -9.111, -149.935, 51.835, 160.318]
  Set speed (17.5 mm/s)
  Call Extruder(89.23980)
  MoveL 9562 to (531.93, 479.33, 172) mm, rotated rx -180 ry 0 rz 160 deg; joints [3.365, 57.073, -9.498, -149.661, 51.734, 160.077]
  Call Extruder(93.33692)
  MoveL 9563 to (532.59, 480.41, 172) mm, rotated rx -180 ry 0 rz 160 deg; joints [3.488, 57.211, -9.76, -149.465, 51.67, 159.906]
  Set speed (17.5 mm/s)
  Call Extruder(95.85107)
  MoveL 9564 to (532.99, 481.08, 172) mm, rotated rx 180 ry 0 rz 160 deg; joints [3.564, 57.294, -9.917, -149.344, 51.633, 159.801]
  Call Extruder(98.47164)
  MoveL 9565 to (533.39, 481.79, 172) mm, rotated rx -180 ry 0 rz 160 deg; joints [3.645, 57.378, -10.075, -149.217, 51.597, 159.693]
  Call Extruder(101.30261)
  MoveL 9566 to (533.8, 482.57, 172) mm, rotated rx 180 ry 0 rz 160 deg; joints [3.734, 57.466, -10.241, -149.079, 51.561, 159.576]
  Set speed (17.5 mm/s)
  Call Extruder(105.66872)
  MoveL 9567 to (534.4, 483.78, 172) mm, rotated rx -180 ry 0 rz 160 deg; joints [3.872, 57.596, -10.486, -148.867, 51.511, 159.397]
  Set speed (17.5 mm/s)
  Call Extruder(108.69517)
  MoveL 9568 to (534.78, 484.63, 172) mm, rotated rx 180 ry 0 rz 160 deg; joints [3.969, 57.681, -10.647, -148.719, 51.48, 159.275]
  Set speed (17.5 mm/s)
  Call Extruder(113.51332)
  MoveL 9569 to (535.36, 486.01, 172) mm, rotated rx 180 ry 0 rz 160 deg; joints [4.126, 57.811, -10.891, -148.484, 51.438, 159.081]
  Set speed (17.5 mm/s)
  Call Extruder(118.53928)
  MoveL 9570 to (535.9, 487.46, 172) mm, rotated rx -180 ry 0 rz 160 deg; joints [4.293, 57.936, -11.128, -148.238, 51.403, 158.882]
  Call Extruder(123.53271)
  MoveL 9571 to (536.38, 488.93, 172) mm, rotated rx -180 ry 0 rz 160 deg; joints [4.461, 58.05, -11.343, -147.995, 51.378, 158.689]
  Set speed (17.5 mm/s)
  Call Extruder(128.42788)
  MoveL 9572 to (536.79, 490.39, 172) mm, rotated rx 180 ry 0 rz 160 deg; joints [4.628, 58.152, -11.537, -147.757, 51.362, 158.503]
  Set speed (17.5 mm/s)
  Call Extruder(133.56964)
  MoveL 9573 to (537.16, 491.94, 172) mm, rotated rx -180 ry 0 rz 160 deg; joints [4.806, 58.249, -11.718, -147.509, 51.355, 158.312]
  Call Extruder(138.65922)
  MoveL 9574 to (537.47, 493.49, 172) mm, rotated rx 180 ry 0 rz 160 deg; joints [4.983, 58.333, -11.878, -147.265, 51.358, 158.128]
  Set speed (17.5 mm/s)
  Call Extruder(143.59756)
  MoveL 9575 to (537.7, 495, 172) mm, rotated rx 180 ry 0 rz 160 deg; joints [5.157, 58.405, -12.013, -147.031, 51.37, 157.955]
  Set speed (17.5 mm/s)
  Call Extruder(148.53610)
  MoveL 9576 to (537.87, 496.52, 172) mm, rotated rx 180 ry 0 rz 160 deg; joints [5.333, 58.465, -12.126, -146.8, 51.391, 157.788]
  Set speed (17.5 mm/s)
  Call Extruder(153.72841)
  MoveL 9577 to (537.98, 498.12, 172) mm, rotated rx 180 ry 0 rz 160 deg; joints [5.519, 58.517, -12.225, -146.56, 51.422, 157.618]
  Set speed (17.5 mm/s)
  Call Extruder(158.69547)
  MoveL 9578 to (538.03, 499.66, 172) mm, rotated rx -180 ry 0 rz 160 deg; joints [5.697, 58.555, -12.297, -146.334, 51.462, 157.463]
  Set speed (17.5 mm/s)
  Call Extruder(163.99259)
  MoveL 9579 to (538.01, 501.3, 172) mm, rotated rx 180 ry 0 rz 160 deg; joints [5.888, 58.584, -12.351, -146.097, 51.515, 157.305]
  Set speed (17.5 mm/s)
  Call Extruder(168.79439)
  MoveL 9580 to (537.93, 502.78, 172) mm, rotated rx 180 ry 0 rz 160 deg; joints [6.062, 58.598, -12.378, -145.887, 51.571, 157.168]
  Set speed (17.5 mm/s)
  Call Extruder(173.72407)
  MoveL 9581 to (537.78, 504.3, 172) mm, rotated rx -180 ry 0 rz 160 deg; joints [6.24, 58.603, -12.386, -145.676, 51.638, 157.035]
  Set speed (17.5 mm/s)
  Call Extruder(178.94019)
  MoveL 9582 to (537.57, 505.9, 172) mm, rotated rx 180 ry 0 rz 160 deg; joints [6.429, 58.595, -12.372, -145.457, 51.717, 156.903]
  Set speed (17.5 mm/s)
  Call Extruder(183.85407)
  MoveL 9583 to (537.3, 507.4, 172) mm, rotated rx -180 ry 0 rz 160 deg; joints [6.607, 58.576, -12.337, -145.257, 51.8, 156.786]
  Set speed (17.5 mm/s)
  Call Extruder(189.15196)
  MoveL 9584 to (536.95, 509, 172) mm, rotated rx 180 ry 0 rz 160 deg; joints [6.798, 58.544, -12.276, -145.046, 51.9, 156.669]
  Set speed (17.5 mm/s)
  Call Extruder(194.59265)
  MoveL 9585 to (536.52, 510.63, 172) mm, rotated rx 180 ry 0 rz 160 deg; joints [6.993, 58.499, -12.191, -144.837, 52.01, 156.558]
  Call Extruder(198.86862)
  MoveL 9586 to (536.12, 511.89, 172) mm, rotated rx 180 ry 0 rz 160 deg; joints [7.145, 58.452, -12.102, -144.678, 52.105, 156.479]
  Set speed (17.5 mm/s)
  Call Extruder(201.81457)
  MoveL 9587 to (535.82, 512.76, 172) mm, rotated rx 180 ry 0 rz 160 deg; joints [7.25, 58.415, -12.032, -144.572, 52.173, 156.429]
  Set speed (17.5 mm/s)
  Call Extruder(204.79127)
  MoveL 9588 to (535.51, 513.62, 172) mm, rotated rx 180 ry 0 rz 160 deg; joints [7.355, 58.375, -11.957, -144.466, 52.244, 156.38]
  Set speed (17.5 mm/s)
  Call Extruder(209.22820)
  MoveL 9589 to (534.99, 514.89, 172) mm, rotated rx 180 ry 0 rz 160 deg; joints [7.511, 58.308, -11.83, -144.312, 52.355, 156.314]
  Set speed (17.5 mm/s)
  Call Extruder(213.92502)
  MoveL 9590 to (534.4, 516.22, 172) mm, rotated rx -180 ry 0 rz 160 deg; joints [7.675, 58.227, -11.677, -144.155, 52.479, 156.251]
  Set speed (17.5 mm/s)
  Call Extruder(219.12371)
  MoveL 9591 to (533.68, 517.66, 172) mm, rotated rx -180 ry 0 rz 160 deg; joints [7.854, 58.127, -11.488, -143.989, 52.624, 156.192]
  Set speed (17.5 mm/s)
  Call Extruder(221.57634)
  MoveL 9592 to (533.32, 518.33, 172) mm, rotated rx 180 ry 0 rz 160 deg; joints [7.937, 58.075, -11.39, -143.913, 52.695, 156.168]
  Set speed (17.5 mm/s)
  Call Extruder(225.00620)
  MoveL 9593 to (532.79, 519.25, 172) mm, rotated rx -180 ry 0 rz 160 deg; joints [8.054, 57.999, -11.247, -143.81, 52.796, 156.136]
  Set speed (17.5 mm/s)
  Call Extruder(229.21182)
  MoveL 9594 to (532.11, 520.37, 172) mm, rotated rx -180 ry 0 rz 160 deg; joints [8.195, 57.9, -11.059, -143.688, 52.924, 156.104]
  Set speed (17.5 mm/s)
  Call Extruder(234.04994)
  MoveL 9595 to (531.29, 521.62, 172) mm, rotated rx 180 ry 0 rz 160 deg; joints [8.354, 57.776, -10.827, -143.554, 53.077, 156.076]
  Set speed (17.5 mm/s)
  Call Extruder(236.81577)
  MoveL 9596 to (530.79, 522.31, 172) mm, rotated rx 180 ry 0 rz 160 deg; joints [8.444, 57.702, -10.686, -143.481, 53.167, 156.063]
  Set speed (17.5 mm/s)
  Call Extruder(241.66825)
  MoveL 9597 to (529.89, 523.51, 172) mm, rotated rx -180 ry 0 rz 160 deg; joints [8.6, 57.564, -10.426, -143.357, 53.328, 156.047]
  Call Extruder(244.08644)
  MoveL 9598 to (529.42, 524.1, 172) mm, rotated rx 180 ry 0 rz 160 deg; joints [8.677, 57.492, -10.29, -143.298, 53.411, 156.043]
  Call Extruder(246.64645)
  MoveL 9599 to (528.91, 524.71, 172) mm, rotated rx -180 ry 0 rz 160 deg; joints [8.757, 57.414, -10.142, -143.238, 53.499, 156.04]
  Call Extruder(249.17942)
  MoveL 9600 to (528.39, 525.3, 172) mm, rotated rx 180 ry 0 rz 160 deg; joints [8.836, 57.334, -9.991, -143.18, 53.588, 156.04]
  Set speed (17.5 mm/s)
  Call Extruder(251.61970)
  MoveL 9601 to (527.89, 525.86, 172) mm, rotated rx 180 ry 0 rz 160 deg; joints [8.911, 57.255, -9.842, -143.126, 53.674, 156.042]
  Set speed (17.5 mm/s)
  Call Extruder(254.18169)
  MoveL 9602 to (527.34, 526.43, 172) mm, rotated rx -180 ry 0 rz 160 deg; joints [8.988, 57.169, -9.681, -143.071, 53.766, 156.046]
  Set speed (17.5 mm/s)
  Call Extruder(256.68298)
  MoveL 9603 to (526.8, 526.98, 172) mm, rotated rx -180 ry 0 rz 160 deg; joints [9.063, 57.084, -9.519, -143.02, 53.857, 156.053]
  Set speed (17.5 mm/s)
  Call Extruder(259.21973)
  MoveL 9604 to (526.23, 527.53, 172) mm, rotated rx -180 ry 0 rz 160 deg; joints [9.138, 56.995, -9.352, -142.97, 53.951, 156.062]
  Call Extruder(261.64557)
  MoveL 9605 to (525.69, 528.04, 172) mm, rotated rx -180 ry 0 rz 160 deg; joints [9.208, 56.908, -9.188, -142.924, 54.041, 156.072]
